// NeuroPLC — Auto-generated IEC 61131-3 SCL
// Graph: kan | Target: S71200Backend
// Work memory: 75KB | LUT points: 15
// Nodes: 11 | Ops: {'matmul': 3, 'standard_act': 2, 'bspline_lut': 2, 'add': 2, 'softmax': 1, 'argmax': 1}


DATA_BLOCK "NeuroPLC_Weights"
{ S7_Optimized_Access := 'FALSE' }
VERSION : 0.1
NON_RETAIN
   STRUCT

   // BsplineLUT 'l0_bspline': grid(15 pts) + table(16×28×15)
   w0 : ARRAY[0..14] OF REAL :=
[-3.0000000, -2.5714286, -2.1428571, -1.7142857, -1.2857143, -0.8571429, -0.4285714, 0.0
    0.4285714, 0.8571429, 1.2857143, 1.7142857, 2.1428571, 2.5714286, 3.0000000];
   w1 : ARRAY[0..6719] OF REAL :=
[-0.1678985, -0.1780923, -0.1814521, -0.1775268, -0.1656160, -0.1449310, -0.1146830, -0.0740834
    -0.0224071, 0.0378880, 0.0997435, 0.1557420, 0.1984661, 0.2204984, 0.2159406, -0.0068030
    -0.0092832, -0.0059920, 0.0046129, 0.0216460, 0.0433637, 0.0680215, 0.0938751, 0.1191888
    0.1426669, 0.1636497, 0.1815270, 0.1956886, 0.2055246, 0.2105588, -0.1221549, -0.1171233
    -0.0966766, -0.0587330, -0.0074782, 0.0506872, 0.1093601, 0.1621373, 0.2026832, 0.2280267
    0.2400602, 0.2410554, 0.2332843, 0.2190189, 0.2004736, -0.1071566, -0.1184995, -0.1260945
    -0.1291901, -0.1269063, -0.1183174, -0.1024977, -0.0785217, -0.0455032, -0.0045367, 0.0404215
    0.0851916, 0.1255936, 0.1574478, 0.1771163, -0.2579331, -0.2737922, -0.2772716, -0.2656087
    -0.2406511, -0.2058749, -0.1647583, -0.1207793, -0.0773919, -0.0368323, 0.0004230, 0.0340346
    0.0636633, 0.0889699, 0.1095319, -0.0785050, -0.0811057, -0.0777832, -0.0686172, -0.0542267
    -0.0354211, -0.0130104, 0.0121958, 0.0393740, 0.0670212, 0.0926518, 0.1137036, 0.1276142
    0.1318216, 0.1243265, 0.1783668, 0.2024992, 0.2205571, 0.2295309, 0.2281837, 0.2159047
    0.1920838, 0.1561110, 0.1074165, 0.0474421, -0.0194626, -0.0887214, -0.1557577, -0.2159953
    -0.2651629, -0.0098763, -0.0567750, -0.0900950, -0.1037325, -0.0997373, -0.0830403, -0.0585757
    -0.0312776, -0.0060409, 0.0142129, 0.0294136, 0.0397139, 0.0452663, 0.0462234, 0.0427955
    -0.1445924, -0.1514427, -0.1456748, -0.1261707, -0.0959553, -0.0595173, -0.0213470, 0.0140651
    0.0422729, 0.0610472, 0.0713624, 0.0744433, 0.0715144, 0.0638003, 0.0524706, 0.0649802
    0.0350223, 0.0192966, 0.0229814, 0.0440583, 0.0779662, 0.1201407, 0.1660179, 0.2110452
    0.2512608, 0.2835559, 0.3048884, 0.3122162, 0.3024972, 0.2736655, 0.2887279, 0.2531290
    0.2083726, 0.1575631, 0.1047861, 0.0544741, 0.0110598, -0.0210238, -0.0374280, -0.0380050
    -0.0286788, -0.0158475, -0.0059090, -0.0052614, -0.0190888, 0.0978082, 0.0375382, -0.0283595
    -0.0966197, -0.1622492, -0.2196440, -0.2631995, -0.2873112, -0.2864807, -0.2605327, -0.2169844
    -0.1639538, -0.1095588, -0.0619172, -0.0280842, 0.3787996, 0.3042307, 0.2275823, 0.1533788
    0.0834056, 0.0184802, -0.0405809, -0.0929614, -0.1378582, -0.1751406, -0.2056495, -0.2303015
    -0.2500134, -0.2657017, -0.2780562, 0.1412515, 0.1458592, 0.1559898, 0.1722250, 0.1933805
    0.2176485, 0.2432202, 0.2682872, 0.2910532, 0.3103575, 0.3259565, 0.3376784, 0.3453514
    0.3488037, 0.3478512, 0.0779829, 0.0010007, -0.0646528, -0.1104959, -0.1384850, -0.1542647
    -0.1634839, -0.1717914, -0.1847575, -0.2040232, -0.2255503, -0.2448578, -0.2574643, -0.2588886
    -0.2455201, -0.0444734, -0.0539526, -0.0628650, -0.0722421, -0.0807835, -0.0863650, -0.0868614
    -0.0801473, -0.0641548, -0.0396736, -0.0116243, 0.0147505, 0.0342076, 0.0415045, 0.0324876
    -0.0761592, -0.0368462, 0.0081775, 0.0553801, 0.1025478, 0.1479322, 0.1897853, 0.2263595
    0.2559171, 0.2772311, 0.2898127, 0.2932306, 0.2870536, 0.2708503, 0.2446318, 0.0232008
    0.0053789, -0.0155840, -0.0376546, -0.0582679, -0.0746713, -0.0841116, -0.0838361, -0.0711388
    -0.0456730, -0.0105014, 0.0310470, 0.0756434, 0.1199589, 0.1607804, 0.3611427, 0.2999726
    0.2319509, 0.1606371, 0.0886557, 0.0183016, -0.0481310, -0.1083478, -0.1600664, -0.2015907
    -0.2320727, -0.2507303, -0.2567816, -0.2494446, -0.2283804, 0.2381873, 0.2065935, 0.1685599
    0.1238492, 0.0745029, 0.0233678, -0.0267086, -0.0728783, -0.1123279, -0.1439519, -0.1691131
    -0.1893671, -0.2062695, -0.2213760, -0.2358772, -0.2661355, -0.2041683, -0.1454980, -0.0950915
    -0.0516159, -0.0115122, 0.0287810, 0.0728252, 0.1241262, 0.1833983, 0.2473215, 0.3122611
    0.3745819, 0.4306494, 0.4769619, -0.0463834, -0.0837121, -0.1064505, -0.1077356, -0.0899888
    -0.0589119, -0.0202105, 0.0204099, 0.0572939, 0.0873028, 0.1109346, 0.1289717, 0.1421960
    0.1513896, 0.1572272, -0.0369839, 0.0175120, 0.0567876, 0.0736601, 0.0717070, 0.0583079
    0.0408467, 0.0267074, 0.0231900, 0.0333957, 0.0543573, 0.0826338, 0.1147841, 0.1473674
    0.1771034, 0.0579601, 0.0613396, 0.0567427, 0.0438791, 0.0253106, 0.0046067, -0.0146619
    -0.0289245, -0.0346569, -0.0306635, -0.0191136, -0.0024393, 0.0169272, 0.0365540, 0.0541844
    0.2344523, 0.1852709, 0.1321315, 0.0796445, 0.0306498, -0.0126383, -0.0480064, -0.0732409
    -0.0861622, -0.0862884, -0.0755912, -0.0562338, -0.0303795, -0.0001915, 0.0321418, -0.3219349
    -0.2878197, -0.2440139, -0.1914641, -0.1323293, -0.0691967, -0.0046544, 0.0587098, 0.1183154
    0.1719484, 0.2179248, 0.2546021, 0.2803375, 0.2934885, 0.2928481, 0.1365492, 0.0991861
    0.0671679, 0.0442195, 0.0300286, 0.0228570, 0.0209643, 0.0226107, 0.0260721, 0.0304366
    0.0359652, 0.0430108, 0.0519260, 0.0630637, 0.0765354, 0.2151295, 0.2080802, 0.1835975
    0.1377589, 0.0763824, 0.0087284, -0.0559392, -0.1083561, -0.1393775, -0.1458259, -0.1331474
    -0.1074616, -0.0748881, -0.0415463, -0.0129262, -0.1535066, -0.1489179, -0.1361766, -0.1134237
    -0.0816039, -0.0426522, 0.0014951, 0.0489018, 0.0976467, 0.1465670, 0.1955956, 0.2447508
    0.2940510, 0.3435148, 0.3928187, -0.1842766, -0.1725566, -0.1530151, -0.1261257, -0.0929481
    -0.0547494, -0.0127967, 0.0316428, 0.0773057, 0.1231240, 0.1683109, 0.2121023, 0.2537336
    0.2924404, 0.3273210, -0.3537021, -0.3697125, -0.3730848, -0.3618120, -0.3364379, -0.2984076
    -0.2491672, -0.1901629, -0.1228470, -0.0489823, 0.0292201, 0.1095140, 0.1896530, 0.2673912
    0.3403057, 0.0691459, 0.0560939, 0.0299653, -0.0117787, -0.0650165, -0.1232729, -0.1800701
    -0.2289302, -0.2634472, -0.2808101, -0.2834036, -0.2740183, -0.2554445, -0.2304725, -0.2017861
    0.3468476, 0.3770096, 0.3880946, 0.3739721, 0.3370012, 0.2825406, 0.2159522, 0.1425982
    0.0678194, -0.0041134, -0.0704748, -0.1286606, -0.1760661, -0.2100872, -0.2284960, -0.0560788
    -0.0071707, 0.0405771, 0.0816977, 0.1138511, 0.1358018, 0.1463158, 0.1441588, 0.1281473
    0.0996185, 0.0635531, 0.0252163, -0.0101268, -0.0372110, -0.0516493, -0.3198017, -0.3047755
    -0.2896692, -0.2776229, -0.2658188, -0.2493332, -0.2232402, -0.1826140, -0.1226357, -0.0438484
    0.0454563, 0.1363818, 0.2200311, 0.2875079, 0.3310730, 0.2163881, 0.2115666, 0.1936969
    0.1613140, 0.1183200, 0.0705138, 0.0236961, -0.0163320, -0.0438224, -0.0556595, -0.0525330
    -0.0354296, -0.0053362, 0.0367607, 0.0893699, -0.2378380, -0.2452140, -0.2327680, -0.1957328
    -0.1394797, -0.0729626, -0.0051392, 0.0550326, 0.0987072, 0.1226663, 0.1318229, 0.1317253
    0.1279218, 0.1259604, 0.1306052, -0.2589217, -0.2554902, -0.2427067, -0.2166298, -0.1778840
    -0.1287070, -0.0713383, -0.0080176, 0.0590193, 0.1277189, 0.1962919, 0.2629692, 0.3259821
    0.3835616, 0.4338699, -0.4825098, -0.4378357, -0.3795550, -0.3085476, -0.2284881, -0.1440391
    -0.0598640, 0.0193734, 0.0890515, 0.1466455, 0.1926608, 0.2278395, 0.2529236, 0.2686552
    0.2757685, 0.0510817, 0.0267852, 0.0115559, 0.0100124, 0.0199990, 0.0369665, 0.0563629
    0.0736359, 0.0842873, 0.0865004, 0.0823345, 0.0741517, 0.0643138, 0.0551828, 0.0488068
    -0.3000423, -0.2227166, -0.1399772, -0.0564061, 0.0242198, 0.0984080, 0.1626662, 0.2135022
    0.2474917, 0.2646081, 0.2697350, 0.2681393, 0.2650878, 0.2658477, 0.2746548, -0.3707289
    -0.3179955, -0.2547265, -0.1827821, -0.1066126, -0.0315833, 0.0369392, 0.0935883, 0.1330773
    0.1541022, 0.1611157, 0.1590200, 0.1527170, 0.1471089, 0.1463268, -0.0303282, -0.0316194
    -0.0313303, -0.0258615, -0.0176743, -0.0113720, -0.0115601, -0.0228442, -0.0497415, -0.0923469
    -0.1443644, -0.1989989, -0.2494552, -0.2889386, -0.3116082, 0.1333115, 0.1672112, 0.1852771
    0.1834520, 0.1631691, 0.1278019, 0.0807259, 0.0253167, -0.0350523, -0.0971276, -0.1578280
    -0.2140861, -0.2628341, -0.3010046, -0.3259561, 0.3146413, 0.2845448, 0.2375658, 0.1752124
    0.1014613, 0.0211616, -0.0608367, -0.1396836, -0.2105710, -0.2707883, -0.3206561, -0.3607319
    -0.3915728, -0.4137364, -0.4276623, -0.2953075, -0.2395135, -0.1840440, -0.1340918, -0.0906518
    -0.0532361, -0.0213547, 0.0054823, 0.0277453, 0.0449382, 0.0551681, 0.0564328, 0.0467301
    0.0240579, -0.0127231, -0.3443950, -0.2914325, -0.2230571, -0.1379327, -0.0423431, 0.0547353
    0.1443230, 0.2174405, 0.2652062, 0.2836330, 0.2758078, 0.2453697, 0.1959578, 0.1312112
    0.0552579, -0.5969847, -0.5568496, -0.4988820, -0.4225912, -0.3306850, -0.2270015, -0.1153800
    0.0003402, 0.1162943, 0.2273436, 0.3265080, 0.4066636, 0.4606866, 0.4814535, 0.4636622
    0.4240763, 0.3780873, 0.3254954, 0.2679662, 0.2064849, 0.1417967, 0.0746462, 0.0057781
    -0.0640220, -0.1319213, -0.1921286, -0.2386218, -0.2653784, -0.2663764, -0.2372068, 0.3549311
    0.2616640, 0.1653353, 0.0727070, -0.0142901, -0.0954316, -0.1704954, -0.2392592, -0.3014889
    -0.3563516, -0.4021494, -0.4371169, -0.4594885, -0.4674988, -0.4598311, 0.2618391, 0.2260382
    0.1761623, 0.1113720, 0.0344484, -0.0505477, -0.1395543, -0.2285095, -0.3133526, -0.3901000
    -0.4548796, -0.5038275, -0.5330802, -0.5387741, -0.5180939, 0.1146218, 0.0686993, 0.0261798
    -0.0089268, -0.0355121, -0.0534927, -0.0627863, -0.0633110, -0.0549970, -0.0383974, -0.0149654
    0.0137755, 0.0463018, 0.0810901, 0.1164729, 0.0417326, 0.0411822, 0.0355795, 0.0236865
    0.0051303, -0.0201561, -0.0522397, -0.0911871, -0.1370274, -0.1879016, -0.2392222, -0.2861886
    -0.3240004, -0.3478571, -0.3537749, 0.3919963, 0.3451138, 0.2737949, 0.1739022, 0.0532871
    -0.0759618, -0.2017516, -0.3119893, -0.3947308, -0.4454888, -0.4705520, -0.4770510, -0.4721161
    -0.4628775, -0.4554293, -0.0126168, -0.0509731, -0.0831967, -0.1066613, -0.1219576, -0.1308127
    -0.1349550, -0.1361129, -0.1360037, -0.1357924, -0.1358456, -0.1364676, -0.1379626, -0.1406350
    -0.1446051, 0.2584295, 0.1992141, 0.1407706, 0.0851690, 0.0331316, -0.0150953, -0.0592658
    -0.0991342, -0.1344641, -0.1654932, -0.1931442, -0.2183931, -0.2422161, -0.2655895, -0.2890680
    0.1814504, 0.1560406, 0.1238631, 0.0846020, 0.0413235, -0.0017105, -0.0402371, -0.0699933
    -0.0867895, -0.0901119, -0.0847588, -0.0759432, -0.0688782, -0.0687767, -0.0798079, 0.2167516
    0.2200129, 0.2198452, 0.2137589, 0.2003766, 0.1787147, 0.1477895, 0.1066176, 0.0542793
    -0.0069583, -0.0702222, -0.1282799, -0.1738986, -0.1998461, -0.2001815, 0.3418077, 0.3005003
    0.2533219, 0.2024476, 0.1507898, 0.1015218, 0.0578167, 0.0228482, -0.0002539, -0.0105333
    -0.0101751, -0.0016098, 0.0127324, 0.0304209, 0.0491649, 0.0084501, 0.0182875, 0.0334012
    0.0528385, 0.0750525, 0.0982866, 0.1207838, 0.1407871, 0.1565614, 0.1674692, 0.1744586
    0.1786018, 0.1809709, 0.1826379, 0.1844059, 0.1765064, 0.2196629, 0.2448905, 0.2446444
    0.2216758, 0.1823734, 0.1331302, 0.0803391, 0.0303612, -0.0120419, -0.0444194, -0.0645012
    -0.0700173, -0.0586974, -0.0290885, 0.0325744, -0.0001235, -0.0308025, -0.0574152, -0.0786708
    -0.0935458, -0.1010169, -0.1000610, -0.0896901, -0.0706827, -0.0463699, -0.0202822, 0.0040500
    0.0230964, 0.0337703, -0.0545263, -0.0683008, -0.0850943, -0.1062798, -0.1300055, -0.1532799
    -0.1731101, -0.1865034, -0.1905247, -0.1851252, -0.1744277, -0.1628807, -0.1549326, -0.1550320
    -0.1666709, 0.1232095, 0.0887160, 0.0601212, 0.0408368, 0.0302367, 0.0262682, 0.0268770
    0.0300090, 0.0336161, 0.0359655, 0.0357802, 0.0318186, 0.0228393, 0.0076005, -0.0147278
    0.2201795, 0.2253740, 0.2172903, 0.1919017, 0.1522543, 0.1038936, 0.0523679, 0.0032255
    -0.0380339, -0.0683450, -0.0881606, -0.0982082, -0.0992153, -0.0919093, -0.0771561, -0.0447728
    -0.0640291, -0.0828933, -0.1010502, -0.1166342, -0.1272313, -0.1304274, -0.1238081, -0.1050070
    -0.0740562, -0.0344543, 0.0100294, 0.0556256, 0.0985653, 0.1354940, -0.1179619, -0.0810167
    -0.0497815, -0.0275970, -0.0124455, -0.0004163, 0.0124039, 0.0299280, 0.0560133, 0.0917222
    0.1340779, 0.1797886, 0.2255621, 0.2681066, 0.3042721, -0.1272539, -0.1083060, -0.0797053
    -0.0391874, 0.0101826, 0.0634562, 0.1156826, 0.1619112, 0.1972416, 0.2192794, 0.2292528
    0.2286728, 0.2190502, 0.2018959, 0.1787229, 0.1126120, 0.1354389, 0.1525481, 0.1626929
    0.1662377, 0.1641164, 0.1572638, 0.1466143, 0.1330899, 0.1169858, 0.0976906, 0.0745224
    0.0467991, 0.0138388, -0.0245556, -0.2130979, -0.2165407, -0.2060983, -0.1792987, -0.1401104
    -0.0947774, -0.0495465, -0.0106644, 0.0157041, 0.0274952, 0.0285724, 0.0232618, 0.0158893
    0.0107810, 0.0115579, 0.0891590, 0.1140725, 0.1352188, 0.1521983, 0.1640686, 0.1696956
    0.1679449, 0.1576822, 0.1378004, 0.1085657, 0.0722279, 0.0311922, -0.0121365, -0.0553532
    -0.0961057, 0.1578736, 0.1729503, 0.1827859, 0.1860957, 0.1827528, 0.1730394, 0.1572379
    0.1356310, 0.1085122, 0.0767250, 0.0419077, 0.0057608, -0.0300154, -0.0637205, -0.0937200
    0.1219553, 0.1204909, 0.1111442, 0.0926814, 0.0665890, 0.0353152, 0.0013086, -0.0329816
    -0.0651094, -0.0927796, -0.1139141, -0.1264520, -0.1283324, -0.1174944, -0.0926047, -0.3210574
    -0.2989046, -0.2712918, -0.2394569, -0.2041107, -0.1657779, -0.1249830, -0.0822503, -0.0381294
    0.0055785, 0.0452625, 0.0771708, 0.0975514, 0.1026523, 0.0896807, 0.3200986, 0.2807284
    0.2284062, 0.1641834, 0.0906839, 0.0110872, -0.0714266, -0.1536772, -0.2324955, -0.3052692
    -0.3701901, -0.4255132, -0.4694930, -0.5003846, -0.5167131, -0.1748312, -0.1799129, -0.1605858
    -0.1114278, -0.0414540, 0.0352193, 0.1044700, 0.1521760, 0.1644143, 0.1372339, 0.0810951
    0.0075831, -0.0717166, -0.1452187, -0.2027312, -0.3041509, -0.2639937, -0.2150850, -0.1581814
    -0.0940170, -0.0233181, 0.0531893, 0.1347787, 0.2206823, 0.3080428, 0.3909831, 0.4633908
    0.5191528, 0.5521570, 0.5574339, 0.0965330, 0.0451092, 0.0023842, -0.0276105, -0.0455321
    -0.0536940, -0.0544114, -0.0499998, -0.0427504, -0.0337479, -0.0223328, -0.0077097, 0.0109168
    0.0343421, 0.0629047, -0.0030185, -0.0198640, -0.0314239, -0.0331272, -0.0253625, -0.0102703
    0.0100064, 0.0333250, 0.0575613, 0.0815243, 0.1053716, 0.1293659, 0.1537700, 0.1788468
    0.2045315, -0.3042292, -0.2481812, -0.1946689, -0.1476865, -0.1072513, -0.0719759, -0.0404710
    -0.0113473, 0.0167654, 0.0442961, 0.0703129, 0.0937775, 0.1136519, 0.1288979, 0.1386143
    -0.1048548, -0.1008864, -0.0997962, -0.1004730, -0.1017998, -0.1026578, -0.1019281, -0.0984919
    -0.0912440, -0.0797672, -0.0646386, -0.0465128, -0.0260444, -0.0038881, 0.0191783, -0.0939790
    -0.0398485, 0.0127617, 0.0593301, 0.0980469, 0.1280599, 0.1485184, 0.1585714, 0.1574058
    0.1460905, 0.1284148, 0.1083804, 0.0899891, 0.0772424, 0.0734226, 0.0639287, 0.0862761
    0.0959409, 0.0932695, 0.0824167, 0.0688831, 0.0581708, 0.0557819, 0.0671351, 0.0934834
    0.1300586, 0.1716228, 0.2129377, 0.2487656, 0.2744141, 0.2868718, 0.2211201, 0.1533946
    0.0863596, 0.0213453, -0.0407895, -0.0991865, -0.1529877, -0.2013294, -0.2430814, -0.2767285
    -0.3007249, -0.3135253, -0.3135841, -0.2998512, 0.3022131, 0.2637090, 0.2171172, 0.1644126
    0.1073856, 0.0477614, -0.0127350, -0.0723783, -0.1294486, -0.1824798, -0.2303725, -0.2720563
    -0.3064606, -0.3325149, -0.3492050, 0.3392466, 0.3126993, 0.2714594, 0.2146510, 0.1455293
    0.0688093, -0.0107926, -0.0885596, -0.1597984, -0.2209733, -0.2702214, -0.3058107, -0.3260089
    -0.3290841, -0.3139513, 0.3067191, 0.2591372, 0.2119206, 0.1692937, 0.1304451, 0.0927841
    0.0537179, 0.0106537, -0.0389403, -0.0945411, -0.1512107, -0.2036668, -0.2466268, -0.2748083
    -0.2838474, 0.1625653, 0.1415380, 0.1123944, 0.0749316, 0.0320777, -0.0121329, -0.0536643
    -0.0884808, -0.1126109, -0.1252995, -0.1304398, -0.1322882, -0.1351006, -0.1431335, -0.1597394
    0.5166554, 0.5215591, 0.4949956, 0.4327331, 0.3412310, 0.2307273, 0.1114637, -0.0063177
    -0.1124656, -0.2013636, -0.2739490, -0.3316710, -0.3759787, -0.4083213, -0.4298892, 0.1351729
    0.1269306, 0.1250641, 0.1320221, 0.1440110, 0.1550311, 0.1590802, 0.1501562, 0.1223698
    0.0754777, 0.0173960, -0.0433222, -0.0981235, -0.1384550, -0.1571404, 0.3327708, 0.3185382
    0.3052332, 0.2953537, 0.2875125, 0.2789499, 0.2669047, 0.2486153, 0.2213666, 0.1847521
    0.1417018, 0.0954064, 0.0490564, 0.0058424, -0.0312945, 0.1765392, 0.1838493, 0.1913348
    0.1987953, 0.2042284, 0.2049950, 0.1984554, 0.1819698, 0.1529608, 0.1119811, 0.0641066
    0.0147661, -0.0306112, -0.0665965, -0.0886083, 0.3272812, 0.3066857, 0.2636611, 0.1950108
    0.1051633, 0.0012415, -0.1096290, -0.2203221, -0.3237405, -0.4142143, -0.4881364, -0.5420610
    -0.5725418, -0.5761332, -0.5504896, 0.2278051, 0.2094044, 0.1705757, 0.1099797, 0.0357921
    -0.0404488, -0.1072012, -0.1529231, -0.1662461, -0.1444863, -0.0975110, -0.0361671, 0.0286983
    0.0862383, 0.1270917, -0.1655097, -0.1719809, -0.1668263, -0.1452783, -0.1086140, -0.0602463
    -0.0035905, 0.0579380, 0.1209348, 0.1825338, 0.2406473, 0.2932485, 0.3383102, 0.3738059
    0.3978944, -0.2981057, -0.2943176, -0.2839422, -0.2664428, -0.2405757, -0.2048473, -0.1577640
    -0.0978318, -0.0236287, 0.0626850, 0.1537709, 0.2418867, 0.3192897, 0.3782378, 0.4121280
    -0.1586868, -0.1489341, -0.1283361, -0.0939585, -0.0484726, 0.0034693, 0.0572128, 0.1081034
    0.1515276, 0.1849213, 0.2086818, 0.2234378, 0.2298178, 0.2284506, 0.2200290, -0.1252231
    -0.0967453, -0.0594933, -0.0122600, 0.0401879, 0.0909722, 0.1332126, 0.1600285, 0.1646609
    0.1464161, 0.1133667, 0.0742698, 0.0378823, 0.0129611, 0.0068023, 0.0834799, 0.1379879
    0.1843656, 0.2200514, 0.2444678, 0.2577389, 0.2599891, 0.2513433, 0.2319673, 0.2040831
    0.1728844, 0.1437972, 0.1222471, 0.1136601, 0.1222135, -0.0542189, -0.0593817, -0.0501164
    -0.0211112, 0.0238372, 0.0777129, 0.1334966, 0.1841690, 0.2227778, 0.2457306, 0.2542909
    0.2501011, 0.2348035, 0.2100408, 0.1775758, 0.3034255, 0.2780464, 0.2463558, 0.2100950
    0.1711902, 0.1316324, 0.0934130, 0.0585232, 0.0289297, 0.0053711, -0.0131885, -0.0279235
    -0.0400085, -0.0506181, -0.0606517, -0.3965884, -0.3682756, -0.3285228, -0.2775177, -0.2172121
    -0.1501812, -0.0790007, -0.0062465, 0.0655068, 0.1337557, 0.1960984, 0.2501415, 0.2934912
    0.3237541, 0.3389650, 0.1608326, 0.1162827, 0.0624275, 0.0022430, -0.0599907, -0.1195326
    -0.1716412, -0.2115750, -0.2346503, -0.2390736, -0.2272283, -0.2018240, -0.1655702, -0.1211765
    -0.0713665, -0.3572540, -0.3305627, -0.2893769, -0.2325372, -0.1630612, -0.0854424, -0.0041762
    0.0762423, 0.1513355, 0.2175222, 0.2725155, 0.3141297, 0.3401794, 0.3484788, 0.3373067
    -0.0932589, -0.0570386, -0.0183244, 0.0228229, 0.0646355, 0.1047426, 0.1407726, 0.1703541
    0.1911504, 0.2025709, 0.2065481, 0.2052115, 0.2006907, 0.1951153, 0.1902788, 0.2385926
    0.2339801, 0.2315844, 0.2325340, 0.2356329, 0.2388632, 0.2402064, 0.2376440, 0.2291967
    0.2148689, 0.1975305, 0.1802754, 0.1661975, 0.1583905, 0.1592519, -0.0096166, 0.0259356
    0.0501742, 0.0577008, 0.0510389, 0.0355113, 0.0164439, -0.0008374, -0.0110618, -0.0117129
    -0.0042559, 0.0095336, 0.0278798, 0.0490069, 0.0711183, -0.1487758, -0.1132716, -0.0625716
    0.0072073, 0.0902357, 0.1772524, 0.2589920, 0.3261894, 0.3697036, 0.3866156, 0.3829981
    0.3656259, 0.3412738, 0.3167166, 0.2977738, -0.3100387, -0.2733864, -0.2253677, -0.1644953
    -0.0949510, -0.0229201, 0.0454102, 0.1038525, 0.1462843, 0.1698333, 0.1763237, 0.1679466
    0.1468932, 0.1153546, 0.0757038, -0.1434238, -0.1123590, -0.0765494, -0.0356650, 0.0091617
    0.0562813, 0.1040440, 0.1507999, 0.1949039, 0.2349571, 0.2699162, 0.2987655, 0.3204895
    0.3340726, 0.3386417, -0.5487098, -0.4984198, -0.4303651, -0.3412042, -0.2356422, -0.1212278
    -0.0055129, 0.1039506, 0.1996751, 0.2773809, 0.3374251, 0.3805267, 0.4074045, 0.4187779
    0.4155242, 0.0555172, 0.0089501, -0.0343089, -0.0731426, -0.1051932, -0.1276648, -0.1377611
    -0.1326858, -0.1097181, -0.0699352, -0.0199019, 0.0333883, 0.0829421, 0.1217659, 0.1438930
    0.2507761, 0.2815168, 0.3019036, 0.3074659, 0.2988722, 0.2786065, 0.2491549, 0.2130035
    0.1726394, 0.1305899, 0.0894411, 0.0517834, 0.0202074, -0.0026965, -0.0148557, -0.0135508
    0.0039421, 0.0348047, 0.0815681, 0.1386999, 0.1978184, 0.2505388, 0.2884759, 0.3033705
    0.2932548, 0.2652527, 0.2271982, 0.1869255, 0.1522683, 0.1299458, 0.0477580, 0.0434365
    0.0405601, 0.0394647, 0.0390808, 0.0378424, 0.0341828, 0.0265353, 0.0133655, -0.0052521
    -0.0269176, -0.0490496, -0.0690665, -0.0843869, -0.0928037, -0.0152840, 0.0008645, 0.0171957
    0.0322455, 0.0460338, 0.0591047, 0.0720030, 0.0852735, 0.0994517, 0.1146016, 0.1301063
    0.1452956, 0.1594994, 0.1720476, 0.1822992, 0.0835696, 0.0671618, 0.0535326, 0.0463969
    0.0453883, 0.0486983, 0.0545166, 0.0610332, 0.0664557, 0.0698963, 0.0717732, 0.0726070
    0.0729182, 0.0732271, 0.0737634, 0.1049449, 0.1112980, 0.1163793, 0.1205961, 0.1247603
    0.1298266, 0.1367502, 0.1464860, 0.1599555, 0.1763988, 0.1926262, 0.2052584, 0.2109159
    0.2062195, 0.1885442, 0.2000310, 0.2137095, 0.2303120, 0.2509218, 0.2733334, 0.2941791
    0.3100896, 0.3176959, 0.3136782, 0.2971869, 0.2709424, 0.2379440, 0.2011906, 0.1636813
    0.1281933, 0.1573572, 0.1343969, 0.1147326, 0.1017420, 0.0937354, 0.0872329, 0.0787526
    0.0648123, 0.0420057, 0.0107119, -0.0232191, -0.0535104, -0.0738849, -0.0780657, -0.0611948
    0.3010531, 0.2891479, 0.2765397, 0.2656909, 0.2555265, 0.2437214, 0.2279492, 0.2058837
    0.1752459, 0.1361346, 0.0920856, 0.0469026, 0.0043893, -0.0316503, -0.0579024, 0.1635860
    0.1539574, 0.1472781, 0.1463320, 0.1504416, 0.1577061, 0.1662235, 0.1740918, 0.1794204
    0.1809034, 0.1780789, 0.1705511, 0.1579241, 0.1398021, 0.1161234, 0.0888673, 0.0620743
    0.0338401, 0.0057287, -0.0215293, -0.0474983, -0.0717428, -0.0938275, -0.1133227, -0.1300893
    -0.1444077, -0.1565912, -0.1669530, -0.1758066, -0.1833186, 0.0159197, 0.0066792, 0.0149232
    0.0446014, 0.0900386, 0.1421585, 0.1918811, 0.2301262, 0.2479353, 0.2424391, 0.2195677
    0.1859386, 0.1481690, 0.1128762, 0.0858354, -0.0713168, -0.0199502, 0.0298431, 0.0751292
    0.1142513, 0.1460038, 0.1691816, 0.1825797, 0.1850275, 0.1770806, 0.1617894, 0.1423990
    0.1221546, 0.1043013, 0.0916331, -0.0334748, -0.0320376, -0.0298014, -0.0261495, -0.0216799
    -0.0174198, -0.0143968, -0.0136387, -0.0161503, -0.0218034, -0.0288312, -0.0353396, -0.0394340
    -0.0392202, -0.0331915, 0.1773249, 0.1659503, 0.1539691, 0.1420005, 0.1311617, 0.1227461
    0.1180473, 0.1183589, 0.1249412, 0.1373938, 0.1529160, 0.1685197, 0.1812167, 0.1880190
    0.1864402, -0.2923942, -0.2707606, -0.2375588, -0.1917769, -0.1361762, -0.0748510, -0.0118972
    0.0485893, 0.1025440, 0.1474720, 0.1831465, 0.2095181, 0.2265374, 0.2341547, 0.2324708
    -0.0474071, 0.0251755, 0.0902499, 0.1411504, 0.1772774, 0.2001740, 0.2113859, 0.2124588
    0.2049538, 0.1912038, 0.1746566, 0.1588474, 0.1473110, 0.1435826, 0.1502753, 0.1321979
    0.1203561, 0.1131415, 0.1109601, 0.1125794, 0.1161880, 0.1199738, 0.1221245, 0.1208447
    0.1151616, 0.1052926, 0.0915474, 0.0742361, 0.0536686, 0.0303347, 0.0827111, 0.0475570
    0.0205481, 0.0064576, 0.0037487, 0.0086548, 0.0174068, 0.0262355, 0.0314206, 0.0316776
    0.0292422, 0.0266253, 0.0263375, 0.0308897, 0.0422453, 0.1559601, 0.1618557, 0.1639675
    0.1625987, 0.1582690, 0.1515748, 0.1431125, 0.1334783, 0.1232918, 0.1143282, 0.1100325
    0.1139804, 0.1297475, 0.1609094, 0.2098307, 0.1285062, 0.1413710, 0.1501217, 0.1516426
    0.1458683, 0.1338110, 0.1164840, 0.0949008, 0.0700792, 0.0432541, 0.0159743, -0.0101868
    -0.0336558, -0.0528596, -0.0664548, 0.0948606, 0.1268761, 0.1429078, 0.1405430, 0.1236279
    0.0982197, 0.0703786, 0.0461643, 0.0315498, 0.0281420, 0.0312390, 0.0356463, 0.0361692
    0.0276133, 0.0058732, 0.0552858, 0.0502080, 0.0525088, 0.0651903, 0.0857229, 0.1096220
    0.1324009, 0.1495731, 0.1567168, 0.1526599, 0.1409268, 0.1254085, 0.1099961, 0.0985806
    0.0943855, 0.0418396, 0.0817039, 0.1172940, 0.1463238, 0.1689135, 0.1860333, 0.1986548
    0.2077493, 0.2142760, 0.2185863, 0.2201529, 0.2183801, 0.2126721, 0.2024331, 0.1872655
    0.4663633, 0.4355268, 0.3870336, 0.3232322, 0.2491057, 0.1705683, 0.0935353, 0.0239218
    -0.0324135, -0.0724439, -0.0972354, -0.1081735, -0.1066439, -0.0940319, -0.0719729, 0.0738696
    0.0965428, 0.1211297, 0.1485437, 0.1765138, 0.2016438, 0.2205362, 0.2297934, 0.2260842
    0.2093901, 0.1844801, 0.1564972, 0.1305842, 0.1118842, 0.1046228, 0.1359003, 0.1015587
    0.0673522, 0.0339288, 0.0038379, -0.0196987, -0.0334586, -0.0342193, -0.0188388, 0.0118115
    0.0510589, 0.0917779, 0.1268432, 0.1491292, 0.1527306, -0.1220373, -0.0604971, -0.0028596
    0.0487916, 0.0932368, 0.1295615, 0.1568516, 0.1741927, 0.1807054, 0.1772387, 0.1671403
    0.1539529, 0.1412190, 0.1324815, 0.1306253, 0.0507799, 0.0258565, -0.0043974, -0.0401240
    -0.0786176, -0.1161662, -0.1490565, -0.1735753, -0.1860673, -0.1857758, -0.1761328, -0.1608979
    -0.1438302, -0.1286890, -0.1186756, 0.2325362, 0.2295055, 0.2162579, 0.1904587, 0.1550309
    0.1147558, 0.0744166, 0.0387964, 0.0126389, -0.0013057, -0.0031671, 0.0066999, 0.0279406
    0.0602003, 0.1026374, 0.1164177, 0.0673135, 0.0136762, -0.0426207, -0.0976070, -0.1465717
    -0.1848031, -0.2075894, -0.2102974, -0.1922244, -0.1583484, -0.1140907, -0.0648728, -0.0161160
    0.0272466, 0.1381471, 0.1253827, 0.1192710, 0.1220552, 0.1312882, 0.1428656, 0.1526812
    0.1566288, 0.1506559, 0.1334072, 0.1074253, 0.0755570, 0.0406492, 0.0055486, -0.0271285
    0.0680312, 0.0441387, 0.0219850, 0.0050373, -0.0067235, -0.0145474, -0.0196863, -0.0233920
    -0.0268993, -0.0306000, -0.0336679, -0.0351812, -0.0342186, -0.0298583, -0.0212543, 0.0143462
    0.0564369, 0.0923979, 0.1172092, 0.1314177, 0.1375374, 0.1380842, 0.1355744, 0.1324771
    0.1289144, 0.1216162, 0.1070474, 0.0816731, 0.0419583, -0.0146039, 0.0458034, 0.0375886
    0.0329915, 0.0328845, 0.0373095, 0.0460150, 0.0587492, 0.0752602, 0.0952915, 0.1183475
    0.1435870, 0.1701418, 0.1971439, 0.2237252, 0.2489738, -0.0675705, -0.0779349, -0.0892847
    -0.1018459, -0.1132911, -0.1203910, -0.1199152, -0.1086332, -0.0833887, -0.0447216, 0.0014854
    0.0489326, 0.0913204, 0.1223493, 0.1366654, 0.1363059, 0.1604894, 0.1730149, 0.1692112
    0.1498870, 0.1177873, 0.0756596, 0.0262511, -0.0276837, -0.0830434, -0.1362242, -0.1835831
    -0.2214774, -0.2462641, -0.2549900, -0.0584784, -0.0510379, -0.0453863, -0.0418930, -0.0391219
    -0.0349994, -0.0274510, -0.0144024, 0.0061898, 0.0348083, 0.0696802, 0.1088568, 0.1503891
    0.1923286, 0.2326227, -0.4725194, -0.4550803, -0.4159488, -0.3504955, -0.2650665, -0.1698862
    -0.0751833, 0.0088134, 0.0719969, 0.1103557, 0.1286876, 0.1324779, 0.1272120, 0.1183756
    0.1108190, -0.0580407, -0.0716919, -0.0771220, -0.0708079, -0.0542702, -0.0308122, -0.0037389
    0.0236447, 0.0480749, 0.0683585, 0.0862949, 0.1039172, 0.1232585, 0.1463517, 0.1745565
    -0.1139666, -0.1009195, -0.0615193, 0.0101379, 0.1046543, 0.2072248, 0.3030380, 0.3772829
    0.4153398, 0.4121848, 0.3766607, 0.3186933, 0.2482083, 0.1751314, 0.1084884, -0.3386503
    -0.2988836, -0.2520140, -0.1994287, -0.1442256, -0.0901074, -0.0407772, 0.0000617, 0.0287629
    0.0445271, 0.0506694, 0.0508261, 0.0486337, 0.0477283, 0.0511901, -0.0937131, -0.0158989
    0.0475020, 0.0900333, 0.1133672, 0.1220482, 0.1206241, 0.1136427, 0.1056101, 0.0989486
    0.0930689, 0.0871467, 0.0803574, 0.0718768, 0.0610300, 0.1474761, 0.1859243, 0.2155211
    0.2335537, 0.2385381, 0.2294242, 0.2051623, 0.1647029, 0.1070674, 0.0348320, -0.0442895
    -0.1221825, -0.1907323, -0.2418242, -0.2686586, 0.2542709, 0.2512925, 0.2350916, 0.2048720
    0.1630291, 0.1130858, 0.0585664, 0.0029951, -0.0501248, -0.0983384, -0.1407059, -0.1764061
    -0.2046175, -0.2245187, -0.2353762, -0.2790252, -0.2515094, -0.2084679, -0.1471647, -0.0717860
    0.0110360, 0.0946665, 0.1724704, 0.2378644, 0.2868490, 0.3191584, 0.3348185, 0.3338551
    0.3162940, 0.2826756, 0.2748486, 0.2728063, 0.2621618, 0.2451437, 0.2223791, 0.1939294
    0.1598549, 0.1202163, 0.0751019, 0.0259923, -0.0236204, -0.0700867, -0.1097573, -0.1389828
    -0.1546804, -0.2623799, -0.2054985, -0.1354963, -0.0521019, 0.0400954, 0.1347880, 0.2256666
    0.3064217, 0.3707773, 0.4141263, 0.4342729, 0.4292103, 0.3969309, 0.3354278, 0.2440885
    0.1392560, 0.1162300, 0.0964252, 0.0810994, 0.0696869, 0.0609776, 0.0537605, 0.0468247
    0.0389880, 0.0305027, 0.0236943, 0.0210503, 0.0250582, 0.0382052, 0.0621977, 0.1259315
    0.1096482, 0.0875181, 0.0581287, 0.0236383, -0.0125329, -0.0469632, -0.0762311, -0.0969535
    -0.1076879, -0.1097951, -0.1048552, -0.0944481, -0.0801536, -0.0635219, 0.2101911, 0.1560738
    0.0989987, 0.0431247, -0.0091678, -0.0561267, -0.0960009, -0.1270391, -0.1475136, -0.1568758
    -0.1562811, -0.1470178, -0.1303744, -0.1076393, -0.0802330, -0.0709978, -0.0563350, -0.0357067
    -0.0128466, 0.0108368, 0.0347564, 0.0583261, 0.0809597, 0.1020719, 0.1211274, 0.1376621
    0.1512178, 0.1613361, 0.1675588, 0.1694942, 0.1224296, 0.1043274, 0.0855731, 0.0694867
    0.0561944, 0.0446940, 0.0339819, 0.0230546, 0.0109156, -0.0030746, -0.0190398, -0.0370635
    -0.0572292, -0.0796205, -0.1040558, -0.0767903, -0.1393753, -0.1880802, -0.2176469, -0.2287871
    -0.2243221, -0.2070753, -0.1798703, -0.1455360, -0.1071745, -0.0682824, -0.0323871, -0.0030160
    0.0163035, 0.0227576, -0.0137194, 0.0050569, 0.0242377, 0.0420958, 0.0577960, 0.0708180
    0.0806417, 0.0867471, 0.0886291, 0.0865180, 0.0817078, 0.0755753, 0.0694973, 0.0648508
    0.0627691, 0.5899228, 0.5530820, 0.4900197, 0.3984393, 0.2863394, 0.1653566, 0.0471317
    -0.0566946, -0.1346190, -0.1820228, -0.2042359, -0.2073654, -0.1975180, -0.1808006, -0.1627267
    0.0027698, 0.0031818, 0.0082551, 0.0186404, 0.0351286, 0.0585600, 0.0897753, 0.1296150
    0.1788560, 0.2350957, 0.2913363, 0.3402212, 0.3743939, 0.3864978, 0.3706397, -0.0025321
    0.0205917, 0.0429694, 0.0624773, 0.0793088, 0.0944761, 0.1089923, 0.1238704, 0.1400876
    0.1568265, 0.1706758, 0.1780221, 0.1752515, 0.1587505, 0.1258989, 0.0653871, 0.1041137
    0.1299338, 0.1369698, 0.1280959, 0.1092785, 0.0864875, 0.0656929, 0.0527867, 0.0497712
    0.0530262, 0.0584930, 0.0621127, 0.0598263, 0.0482771, 0.2008938, 0.2139753, 0.2194843
    0.2154537, 0.2038885, 0.1881971, 0.1717893, 0.1580751, 0.1504253, 0.1502483, 0.1561170
    0.1663828, 0.1793971, 0.1935114, 0.2071681, 0.1853853, 0.2319104, 0.2758777, 0.3132807
    0.3417447, 0.3594712, 0.3646623, 0.3555205, 0.3302888, 0.2892609, 0.2356933, 0.1730742
    0.1048913, 0.0346328, -0.0345319, 0.2946110, 0.2887431, 0.2792968, 0.2666786, 0.2517614
    0.2355833, 0.2191820, 0.2035956, 0.1898666, 0.1792673, 0.1734019, 0.1739004, 0.1823929
    0.2005095, 0.2291908, 0.1584648, 0.1666528, 0.1783353, 0.1939631, 0.2109868, 0.2257967
    0.2347820, 0.2343319, 0.2208878, 0.1935178, 0.1550855, 0.1087505, 0.0576728, 0.0050121
    -0.0461847, 0.1433635, 0.1457650, 0.1450598, 0.1404541, 0.1326062, 0.1226875, 0.1118699
    0.1013256, 0.0922152, 0.0851375, 0.0798789, 0.0761625, 0.0737114, 0.0722486, 0.0715160
    0.0642120, 0.0710823, 0.0799319, 0.0885070, 0.0971988, 0.1073328, 0.1202358, 0.1372344
    0.1596237, 0.1871156, 0.2171343, 0.2469256, 0.2737350, 0.2948082, 0.3077406, 0.0792082
    0.0430626, 0.0187277, 0.0104475, 0.0159365, 0.0306019, 0.0498483, 0.0690801, 0.0837509
    0.0917590, 0.0945363, 0.0937904, 0.0912291, 0.0885601, 0.0872292, -0.0366219, -0.0059975
    0.0211352, 0.0437861, 0.0615249, 0.0741193, 0.0813369, 0.0829455, 0.0787241, 0.0690206
    0.0550045, 0.0379096, 0.0189697, -0.0005816, -0.0195318, 0.1408100, 0.1453754, 0.1567995
    0.1752028, 0.1973212, 0.2186946, 0.2348618, 0.2413613, 0.2338025, 0.2113334, 0.1782158
    0.1391110, 0.0986801, 0.0615845, 0.0318855, 0.3728876, 0.3636605, 0.3531002, 0.3411653
    0.3270430, 0.3096478, 0.2878939, 0.2606955, 0.2269944, 0.1871089, 0.1433476, 0.0981741
    0.0540520, 0.0134451, -0.0214319, 0.2175054, 0.2198412, 0.2244289, 0.2304279, 0.2359889
    0.2389059, 0.2369727, 0.2279830, 0.2097863, 0.1830311, 0.1524101, 0.1229322, 0.0996059
    0.0874400, 0.0903775, 0.2911958, 0.2672293, 0.2417178, 0.2170962, 0.1953312, 0.1782237
    0.1675746, 0.1651847, 0.1727999, 0.1894183, 0.2100667, 0.2294619, 0.2423206, 0.2433596
    0.2283258, 0.3827878, 0.3411886, 0.2981977, 0.2569056, 0.2171632, 0.1776772, 0.1371527
    0.0942950, 0.0478225, -0.0028898, -0.0575175, -0.1156620, -0.1769250, -0.2409081, -0.3066716
    0.2251391, 0.2507458, 0.2758858, 0.2986796, 0.3178295, 0.3322430, 0.3408278, 0.3424918
    0.3361631, 0.3217956, 0.3008249, 0.2748025, 0.2452798, 0.2138081, 0.1819130, 0.1689708
    0.1711256, 0.1707270, 0.1694824, 0.1680544, 0.1667367, 0.1658224, 0.1656048, 0.1663845
    0.1688381, 0.1741858, 0.1836898, 0.1986126, 0.2202167, 0.2490858, 0.1198459, 0.1158715
    0.1187188, 0.1281465, 0.1421744, 0.1582081, 0.1736523, 0.1859118, 0.1924255, 0.1923409
    0.1872750, 0.1790374, 0.1694379, 0.1602861, 0.1530649, 0.2813690, 0.2857699, 0.2775994
    0.2518772, 0.2097207, 0.1544021, 0.0891956, 0.0173756, -0.0577623, -0.1318692, -0.1990736
    -0.2533852, -0.2888138, -0.2993691, -0.2805221, -0.0945949, -0.0859146, -0.0666549, -0.0339619
    0.0098287, 0.0605471, 0.1140217, 0.1660807, 0.2125873, 0.2511515, 0.2819078, 0.3051879
    0.3213233, 0.3306457, 0.3334457, 0.1866198, 0.1884683, 0.1787530, 0.1577976, 0.1277766
    0.0915189, 0.0518542, 0.0116119, -0.0263894, -0.0598831, -0.0874005, -0.1075351, -0.1188804
    -0.1200301, -0.1100685, -0.0816909, -0.0186953, 0.0434542, 0.1009326, 0.1520018, 0.1956610
    0.2309103, 0.2567496, 0.2721971, 0.2771671, 0.2728699, 0.2606167, 0.2417188, 0.2174875
    0.1892796, 0.1155247, 0.1110856, 0.1127015, 0.1249412, 0.1436904, 0.1617671, 0.1719855
    0.1671601, 0.1402411, 0.0909893, 0.0290077, -0.0353323, -0.0916595, -0.1296024, -0.1405761
    0.0366876, 0.0358489, 0.0423771, 0.0582548, 0.0821032, 0.1113558, 0.1434446, 0.1758020
    0.2058747, 0.2318435, 0.2529499, 0.2685182, 0.2778728, 0.2803380, 0.2754306, 0.0936999
    0.0709418, 0.0538988, 0.0490415, 0.0548760, 0.0670938, 0.0813836, 0.0934337, 0.0989831
    0.0962942, 0.0872764, 0.0741241, 0.0590313, 0.0441924, 0.0315632, 0.0454234, 0.0491984
    0.0596057, 0.0783299, 0.1034458, 0.1317532, 0.1600503, 0.1851351, 0.2038397, 0.2146847
    0.2186308, 0.2168294, 0.2104321, 0.2005902, 0.1883695, -0.0667184, -0.0664766, -0.0577000
    -0.0366789, -0.0050464, 0.0336767, 0.0759675, 0.1183029, 0.1571787, 0.1900285, 0.2156412
    0.2329118, 0.2407350, 0.2380057, 0.2240467, -0.2274597, -0.1690933, -0.1114029, -0.0583104
    -0.0110341, 0.0301627, 0.0650176, 0.0932684, 0.1146536, 0.1289366, 0.1359178, 0.1354002
    0.1271870, 0.1110814, 0.0872085, -0.1521940, -0.1380929, -0.1188272, -0.0936891, -0.0636631
    -0.0303315, 0.0047229, 0.0399170, 0.0736799, 0.1050380, 0.1338809, 0.1601658, 0.1838497
    0.2048900, 0.2230166, -0.1046155, -0.0858807, -0.0573247, -0.0168516, 0.0333484, 0.0895709
    0.1481097, 0.2052584, 0.2573313, 0.3016632, 0.3370647, 0.3624612, 0.3767782, 0.3789415
    0.3681934, 0.2072487, 0.1864112, 0.1563267, 0.1171031, 0.0715261, 0.0233276, -0.0237592
    -0.0660013, -0.0997112, -0.1234848, -0.1392170, -0.1490607, -0.1551685, -0.1596933, -0.1644943
    -0.1517255, -0.1193664, -0.0782033, -0.0303212, 0.0200548, 0.0679433, 0.1083623, 0.1363294
    0.1469480, 0.1396034, 0.1198693, 0.0938024, 0.0674594, 0.0468970, 0.0370763, 0.3110608
    0.2861295, 0.2560543, 0.2233990, 0.1888246, 0.1523195, 0.1138714, 0.0734681, 0.0311259
    -0.0117016, -0.0514840, -0.0845288, -0.1071434, -0.1156352, -0.1071404, -0.0434422, -0.0256309
    -0.0061618, 0.0137750, 0.0348048, 0.0581937, 0.0852092, 0.1171182, 0.1551570, 0.1990083
    0.2461095, 0.2937233, 0.3391118, 0.3795376, 0.4124577, 0.3129768, 0.3337277, 0.3466819
    0.3502223, 0.3445130, 0.3303478, 0.3085208, 0.2798265, 0.2450805, 0.2061687, 0.1665232
    0.1296974, 0.0992442, 0.0787167, 0.0710807, -0.1485267, -0.1266887, -0.1059538, -0.0874314
    -0.0694476, -0.0493445, -0.0244634, 0.0078547, 0.0501971, 0.1015688, 0.1557980, 0.2063088
    0.2465250, 0.2698708, 0.2709672, 0.0836342, 0.1186020, 0.1419933, 0.1506651, 0.1472868
    0.1365815, 0.1232745, 0.1120911, 0.1076754, 0.1105969, 0.1155374, 0.1167185, 0.1083621
    0.0846902, 0.0412880, 0.3746155, 0.3008116, 0.2295846, 0.1697616, 0.1228553, 0.0877933
    0.0635006, 0.0489020, 0.0429200, 0.0443591, 0.0518531, 0.0640224, 0.0794876, 0.0968693
    0.1147441, 0.2624251, 0.2889178, 0.2926807, 0.2688918, 0.2221700, 0.1604698, 0.0917496
    0.0239679, -0.0349867, -0.0807150, -0.1138608, -0.1354617, -0.1465550, -0.1481785, -0.1414872
    -0.2038390, -0.1836262, -0.1623666, -0.1409924, -0.1188838, -0.0948732, -0.0677921, -0.0364720
    0.0002305, 0.0422140, 0.0875773, 0.1342791, 0.1802779, 0.2235323, 0.2620180, 0.2164622
    0.2150818, 0.2096564, 0.2016837, 0.1911032, 0.1773035, 0.1596727, 0.1375989, 0.1105010
    0.0793446, 0.0473304, 0.0178336, -0.0057705, -0.0201069, -0.0225886, 0.1444894, 0.1318568
    0.1201072, 0.1098967, 0.1011122, 0.0933685, 0.0862802, 0.0794619, 0.0725155, 0.0644148
    0.0532257, 0.0369429, 0.0135614, -0.0189239, -0.0617012, -0.3946738, -0.3444622, -0.2891815
    -0.2324311, -0.1744639, -0.1143506, -0.0511602, 0.0160378, 0.0881280, 0.1636738, 0.2378847
    0.3057082, 0.3620918, 0.4019832, 0.4212244, -0.3757093, -0.3162996, -0.2499295, -0.1809414
    -0.1102374, -0.0375038, 0.0375741, 0.1153111, 0.1959576, 0.2765333, 0.3493883, 0.4065088
    0.4398806, 0.4414897, 0.4052696, 0.3683745, 0.3139668, 0.2502587, 0.1805291, 0.1085247
    0.0381577, -0.0266595, -0.0820146, -0.1240428, -0.1512654, -0.1656516, -0.1694398, -0.1648687
    -0.1541766, -0.1394859, -0.1072037, -0.0830137, -0.0531947, -0.0165176, 0.0251676, 0.0689225
    0.1118077, 0.1508839, 0.1832300, 0.2068588, 0.2211318, 0.2255158, 0.2194776, 0.2024842
    0.1744064, -0.3319098, -0.3459042, -0.3396719, -0.3077802, -0.2539578, -0.1851701, -0.1083861
    -0.0305750, 0.0413362, 0.1025240, 0.1512056, 0.1858353, 0.2048676, 0.2067567, 0.1907547
    0.4012429, 0.3313338, 0.2576209, 0.1851532, 0.1146888, 0.0454699, -0.0232633, -0.0922704
    -0.1622683, -0.2318351, -0.2964571, -0.3513798, -0.3918482, -0.4131078, -0.4113880, 0.0432662
    0.0463959, 0.0470551, 0.0450016, 0.0397214, 0.0306044, 0.0170404, -0.0015809, -0.0258282
    -0.0542036, -0.0822218, -0.1051644, -0.1183129, -0.1169490, -0.0974791, 0.0945418, 0.0474351
    0.0144671, -0.0002516, 0.0002686, 0.0105011, 0.0249166, 0.0379856, 0.0442405, 0.0413054
    0.0312731, 0.0165850, -0.0003173, -0.0169924, -0.0312270, 0.2655172, 0.1779016, 0.0932373
    0.0169355, -0.0501629, -0.1088321, -0.1598481, -0.2039869, -0.2420160, -0.2742825, -0.3005254
    -0.3204366, -0.3337076, -0.3400303, -0.3391558, 0.2147407, 0.1649244, 0.1186844, 0.0787383
    0.0455533, 0.0188009, -0.0018479, -0.0167224, -0.0261599, -0.0309140, -0.0323391, -0.0318368
    -0.0308084, -0.0306556, -0.0325397, 0.3099983, 0.2146933, 0.1365787, 0.0858170, 0.0575848
    0.0417632, 0.0282275, 0.0068529, -0.0323252, -0.0912628, -0.1603408, -0.2290366, -0.2868275
    -0.3231913, -0.3294227, 0.2400604, 0.2115027, 0.1766969, 0.1370982, 0.0944029, 0.0503929
    0.0068497, -0.0344446, -0.0717136, -0.1034392, -0.1284772, -0.1457126, -0.1540302, -0.1523151
    -0.1398969, -0.3239543, -0.2696758, -0.2072356, -0.1376939, -0.0635290, 0.0122797, 0.0867520
    0.1569077, 0.2197818, 0.2731606, 0.3159163, 0.3470059, 0.3653866, 0.3700153, 0.3602427
    -0.1058964, -0.1240447, -0.1388698, -0.1496570, -0.1540083, -0.1489309, -0.1314311, -0.0985154
    -0.0472808, 0.0206385, 0.0970508, 0.1732528, 0.2405411, 0.2902125, 0.3149041, -0.0809075
    -0.0761908, -0.0678088, -0.0552605, -0.0376747, -0.0140495, 0.0166171, 0.0553272, 0.1030094
    0.1569253, 0.2090360, 0.2508892, 0.2740322, 0.2700127, 0.2324689, 0.0183774, 0.0161987
    0.0196904, 0.0307010, 0.0474037, 0.0666728, 0.0853814, 0.1004023, 0.1086441, 0.1087988
    0.1021359, 0.0901261, 0.0742400, 0.0559482, 0.0367036, -0.0097957, -0.0039892, 0.0028189
    0.0105871, 0.0193478, 0.0291596, 0.0400810, 0.0521704, 0.0654758, 0.0795114, 0.0930206
    0.1046862, 0.1131914, 0.1172192, 0.1157655, 0.1191704, 0.1311087, 0.1458877, 0.1635177
    0.1823133, 0.1999896, 0.2142612, 0.2228424, 0.2234735, 0.2151740, 0.1988128, 0.1754036
    0.1459593, 0.1114936, 0.0729542, 0.1572977, 0.1453381, 0.1355189, 0.1300476, 0.1291831
    0.1324956, 0.1395545, 0.1499293, 0.1631903, 0.1789441, 0.1968503, 0.2165725, 0.2377743
    0.2601195, 0.2829789, 0.0628695, 0.0769969, 0.0860344, 0.0877927, 0.0827342, 0.0722577
    0.0577633, 0.0406512, 0.0223093, 0.0035208, -0.0158050, -0.0358270, -0.0567041, -0.0785953
    -0.1016069, 0.1131401, 0.1069956, 0.0981420, 0.0867915, 0.0734585, 0.0587646, 0.0433313
    0.0277801, 0.0127375, -0.0009211, -0.0119603, -0.0191169, -0.0211274, -0.0167287, -0.0051465
    0.0572075, 0.0357429, 0.0213811, 0.0165095, 0.0211165, 0.0343429, 0.0553284, 0.0832127
    0.1171167, 0.1552116, 0.1942961, 0.2310619, 0.2622007, 0.2844040, 0.2948321, 0.1434070
    0.1549482, 0.1670772, 0.1781332, 0.1874069, 0.1945248, 0.1991140, 0.2008018, 0.1992118
    0.1938003, 0.1837813, 0.1683501, 0.1467019, 0.1180318, 0.0819414, 0.0750777, 0.0777608
    0.0672206, 0.0439258, 0.0107293, -0.0286731, -0.0705851, -0.1113101, -0.1471814, -0.1760247
    -0.1978224, -0.2127253, -0.2208840, -0.2224495, -0.2176575, 0.1612096, 0.1444548, 0.1335241
    0.1296110, 0.1294437, 0.1281723, 0.1209451, 0.1029104, 0.0692988, 0.0194586, -0.0413110
    -0.1072460, -0.1725826, -0.2315571, -0.2789746, 0.4111212, 0.3551752, 0.2895649, 0.2152339
    0.1348414, 0.0516528, -0.0310660, -0.1100489, -0.1820429, -0.2444422, -0.2955766, -0.3338489
    -0.3576620, -0.3654186, -0.3560661, 0.1391590, 0.1250600, 0.1217095, 0.1317212, 0.1507030
    0.1717879, 0.1881056, 0.1927863, 0.1790760, 0.1460479, 0.1011956, 0.0526702, 0.0086227
    -0.0227959, -0.0347899, 0.0559819, 0.0581868, 0.0646391, 0.0766424, 0.0923719, 0.1088978
    0.1232888, 0.1326139, 0.1339891, 0.1269062, 0.1142898, 0.0993324, 0.0852266, 0.0751649
    0.0718163, 0.2732919, 0.2494898, 0.2191522, 0.1815386, 0.1363864, 0.0836023, 0.0230931
    -0.0452346, -0.1214316, -0.2034314, -0.2861067, -0.3640917, -0.4320202, -0.4845264, -0.5169412
    -0.0691999, -0.1076962, -0.1233470, -0.1107835, -0.0727259, -0.0147534, 0.0575521, 0.1386083
    0.2228317, 0.3045648, 0.3780438, 0.4374964, 0.4771504, 0.4912336, 0.4753526, -0.0001498
    -0.0032703, 0.0011039, 0.0176806, 0.0448323, 0.0786930, 0.1153941, 0.1510671, 0.1818855
    0.2061389, 0.2251743, 0.2405776, 0.2539347, 0.2668312, 0.2804183, 0.2785104, 0.2438975
    0.2035888, 0.1580865, 0.1088918, 0.0578585, 0.0068411, -0.0423062, -0.0877313, -0.1277092
    -0.1606971, -0.1851669, -0.1995904, -0.2024393, -0.1926829, 0.4454534, 0.3676981, 0.2863407
    0.2065850, 0.1303759, 0.0585069, -0.0082298, -0.0690421, -0.1231326, -0.1694447, -0.2065468
    -0.2329782, -0.2472781, -0.2479858, -0.2341930, -0.2216615, -0.2067420, -0.1850035, -0.1541864
    -0.1140946, -0.0652607, -0.0082182, 0.0564991, 0.1283061, 0.2040327, 0.2767734, 0.3393309
    0.3845079, 0.4051074, 0.3954616, -0.0241830, -0.0147689, -0.0074899, -0.0015797, 0.0041061
    0.0108452, 0.0199157, 0.0325956, 0.0501315, 0.0722017, 0.0962181, 0.1194157, 0.1390292
    0.1522937, 0.1568849, -0.0959317, -0.0528233, -0.0092763, 0.0343819, 0.0779881, 0.1214369
    0.1646231, 0.2074412, 0.2497654, 0.2904309, 0.3267724, 0.3560070, 0.3753522, 0.3820254
    0.3738285, -0.0641084, -0.0609075, -0.0583547, -0.0550581, -0.0502603, -0.0434279, -0.0340281
    -0.0215279, -0.0054111, 0.0139915, 0.0351259, 0.0563423, 0.0759910, 0.0924222, 0.1041725
    -0.0341204, -0.0091993, 0.0193507, 0.0505301, 0.0828547, 0.1146690, 0.1443173, 0.1701441
    0.1905136, 0.2047915, 0.2137906, 0.2184365, 0.2196550, 0.2183718, 0.2153754, -0.0186932
    0.0193089, 0.0562244, 0.0918554, 0.1257393, 0.1573201, 0.1860417, 0.2113482, 0.2326842
    0.2495404, 0.2614738, 0.2680464, 0.2688202, 0.2633573, 0.2513908, 0.0566885, 0.1031851
    0.1373615, 0.1554016, 0.1597643, 0.1551255, 0.1461639, 0.1375579, 0.1339277, 0.1369582
    0.1440933, 0.1524456, 0.1591280, 0.1612530, 0.1563877, -0.0301588, -0.0067982, 0.0122754
    0.0251599, 0.0333866, 0.0396994, 0.0468439, 0.0575657, 0.0745624, 0.0981387, 0.1251408
    0.1521448, 0.1757269, 0.1924634, 0.1994423, 0.3237398, 0.3147339, 0.2917620, 0.2528614
    0.2016544, 0.1437367, 0.0847061, 0.0301604, -0.0143777, -0.0471586, -0.0718843, -0.0926829
    -0.1136822, -0.1390103, -0.1718136, 0.5322388, 0.4516525, 0.3699894, 0.2936842, 0.2215195
    0.1495740, 0.0739234, -0.0093567, -0.1040900, -0.2090549, -0.3157387, -0.4150598, -0.4979360
    -0.5552858, -0.5795367, 0.3348313, 0.3139692, 0.2890814, 0.2616292, 0.2314300, 0.1977201
    0.1597350, 0.1167106, 0.0679124, 0.0141103, -0.0417528, -0.0965641, -0.1472107, -0.1905800
    -0.2238805, 0.0441595, 0.0223551, 0.0117973, 0.0164633, 0.0346856, 0.0628025, 0.0971498
    0.1340633, 0.1699050, 0.2023456, 0.2309466, 0.2554175, 0.2754675, 0.2908060, 0.3011061
    0.0938526, 0.0646245, 0.0408562, 0.0255288, 0.0176385, 0.0147738, 0.0145215, 0.0144682
    0.0122432, 0.0075938, 0.0033288, 0.0024960, 0.0081430, 0.0233176, 0.0503320, -0.1736872
    -0.2018598, -0.2184409, -0.2198891, -0.2069418, -0.1818479, -0.1468583, -0.1042237, -0.0562133
    -0.0060076, 0.0418950, 0.0828932, 0.1123860, 0.1257721, 0.1194308, 0.2034807, 0.2159660
    0.2251174, 0.2297540, 0.2297332, 0.2252793, 0.2166169, 0.2039706, 0.1875626, 0.1674950
    0.1436959, 0.1160799, 0.0845618, 0.0490560, 0.0097851, 0.0084393, -0.0037575, -0.0096962
    -0.0075738, 0.0020896, 0.0179530, 0.0386746, 0.0629125, 0.0893207, 0.1163582, 0.1422011
    0.1650037, 0.1829203, 0.1941051, 0.1969572, 0.2633480, 0.2195053, 0.1743630, 0.1311768
    0.0902144, 0.0506880, 0.0118084, -0.0272136, -0.0671537, -0.1081212, -0.1492622, -0.1896475
    -0.2283478, -0.2644342, -0.2968259, -0.0753155, -0.0705651, -0.0563480, -0.0336360, -0.0058240
    0.0228373, 0.0480962, 0.0657007, 0.0714666, 0.0645810, 0.0491042, 0.0294766, 0.0101389
    -0.0044685, -0.0106460, 0.2106405, 0.1830579, 0.1505358, 0.1133623, 0.0735978, 0.0339286
    -0.0029582, -0.0343754, -0.0576678, -0.0717680, -0.0779037, -0.0774818, -0.0719092, -0.0625927
    -0.0509060, -0.3274674, -0.2629944, -0.2038490, -0.1565354, -0.1200805, -0.0908690, -0.0652826
    -0.0397029, -0.0105580, 0.0234085, 0.0601056, 0.0971813, 0.1322834, 0.1630599, 0.1873036
    -0.0690877, -0.0509122, -0.0313818, -0.0091832, 0.0158236, 0.0433644, 0.0731640, 0.1049476
    0.1384244, 0.1725134, 0.2049913, 0.2335457, 0.2558642, 0.2696344, 0.2729122, -0.0589441
    -0.0342618, -0.0055190, 0.0271774, 0.0612910, 0.0934264, 0.1201872, 0.1381771, 0.1440491
    0.1369218, 0.1194770, 0.0946747, 0.0654752, 0.0348383, 0.0055348, 0.1142520, 0.1359137
    0.1489129, 0.1481625, 0.1358423, 0.1167002, 0.0954867, 0.0769527, 0.0657870, 0.0635884
    0.0674900, 0.0742760, 0.0807309, 0.0836388, 0.0802503, -0.4963562, -0.4881529, -0.4580787
    -0.4027445, -0.3260558, -0.2344954, -0.1345493, -0.0327034, 0.0645796, 0.1520003, 0.2259398
    0.2829104, 0.3194247, 0.3319951, 0.3183341, -0.2581464, -0.2259318, -0.1867423, -0.1417929
    -0.0931570, -0.0432113, 0.0056672, 0.0511014, 0.0907371, 0.1233640, 0.1494249, 0.1694916
    0.1841360, 0.1939300, 0.1995259, 0.2516904, 0.2530169, 0.2526439, 0.2516513, 0.2490327
    0.2430442, 0.2319413, 0.2139793, 0.1874578, 0.1528830, 0.1139504, 0.0746044, 0.0387894
    0.0104499, -0.0071207, 0.2666245, 0.2363470, 0.2008183, 0.1616806, 0.1188768, 0.0717494
    0.0196403, -0.0381088, -0.1021090, -0.1706225, -0.2385168, -0.3003941, -0.3508568, -0.3845074
    -0.3969070, -0.0286634, -0.0313490, -0.0325963, -0.0315775, -0.0271991, -0.0182737, -0.0036136
    0.0179685, 0.0476130, 0.0841017, 0.1228077, 0.1588378, 0.1872988, 0.2032979, 0.2028342
    0.0822806, 0.1055830, 0.1210727, 0.1261290, 0.1226352, 0.1140661, 0.1038982, 0.0956081
    0.0926303, 0.0963046, 0.1049423, 0.1166188, 0.1294093, 0.1413890, 0.1507615, -0.2690735
    -0.1935901, -0.1172682, -0.0456560, 0.0191559, 0.0762989, 0.1249055, 0.1641084, 0.1930635
    0.2120976, 0.2232291, 0.2286085, 0.2303862, 0.2307129, 0.2313590, -0.0819909, -0.0262301
    0.0238818, 0.0636981, 0.0940510, 0.1177084, 0.1374404, 0.1560169, 0.1761686, 0.1986485
    0.2213520, 0.2419512, 0.2581182, 0.2675254, 0.2681968, -0.0461046, -0.0095733, 0.0161245
    0.0269383, 0.0255286, 0.0169270, 0.0061681, -0.0017138, -0.0017482, 0.0078269, 0.0241367
    0.0439447, 0.0640142, 0.0811086, 0.0923875, 0.1214715, 0.1246429, 0.1179697, 0.1021397
    0.0794863, 0.0529245, 0.0253697, -0.0002625, -0.0210925, -0.0360475, -0.0466648, -0.0546860
    -0.0618522, -0.0699049, -0.0802395, -0.1132871, -0.0717634, -0.0319256, 0.0041296, 0.0359250
    0.0635558, 0.0871177, 0.1067064, 0.1224124, 0.1340688, 0.1411366, 0.1430477, 0.1392339
    0.1291272, 0.1124477, 0.1065226, 0.0679530, 0.0277192, -0.0120758, -0.0494568, -0.0824937
    -0.1092565, -0.1278153, -0.1362775, -0.1346298, -0.1255739, -0.1120240, -0.0968938, -0.0830973
    -0.0731394, 0.0702876, 0.0351664, 0.0094846, -0.0018965, -0.0003208, 0.0106751, 0.0275520
    0.0467709, 0.0648162, 0.0793579, 0.0897788, 0.0955954, 0.0963241, 0.0914817, 0.0808327
    -0.1561871, -0.1465697, -0.1172424, -0.0641265, 0.0073557, 0.0884247, 0.1702974, 0.2441905
    0.3014090, 0.3376742, 0.3550895, 0.3562566, 0.3437775, 0.3202540, 0.2883357, -0.2523765
    -0.2036962, -0.1455273, -0.0788729, -0.0065118, 0.0681494, 0.1417037, 0.2107440, 0.2718817
    0.3226697, 0.3620203, 0.3889524, 0.4024845, 0.4016355, 0.3857890, -0.2730969, -0.2395672
    -0.1975484, -0.1479309, -0.0912749, -0.0280236, 0.0413795, 0.1164914, 0.1968288, 0.2799235
    0.3604371, 0.4328076, 0.4914726, 0.5308703, 0.5462435, 0.2663759, 0.2617837, 0.2487071
    0.2273422, 0.2011032, 0.1745413, 0.1522086, 0.1386574, 0.1383519, 0.1513314, 0.1712411
    0.1912272, 0.2044355, 0.2040123, 0.1844213, -0.1322568, -0.1054526, -0.0694236, -0.0246700
    0.0254581, 0.0766039, 0.1244093, 0.1645163, 0.1926105, 0.2065688, 0.2074343, 0.1964972
    0.1750481, 0.1443772, 0.1058727, 0.0963661, 0.0729697, 0.0442535, 0.0105362, -0.0263189
    -0.0639028, -0.0998057, -0.1316179, -0.1569322, -0.1734747, -0.1791631, -0.1719304, -0.1497096
    -0.1104336, -0.0529810, -0.1897976, -0.1489798, -0.1093301, -0.0766478, -0.0506775, -0.0290246
    -0.0092918, 0.0109181, 0.0339771, 0.0610016, 0.0912931, 0.1240118, 0.1583174, 0.1933700
    0.2281768, -0.0203649, -0.0136181, -0.0048761, 0.0046482, 0.0139614, 0.0221468, 0.0282883
    0.0314697, 0.0308098, 0.0271957, 0.0240692, 0.0250715, 0.0338439, 0.0540278, 0.0882226
    -0.1464982, -0.0937421, -0.0454817, -0.0063742, 0.0244465, 0.0497983, 0.0725012, 0.0953754
    0.1211933, 0.1503596, 0.1798554, 0.2063952, 0.2266930, 0.2374634, 0.2360676, 0.0611053
    0.0746875, 0.0845858, 0.0889394, 0.0865942, 0.0766460, 0.0581907, 0.0303245, -0.0078133
    -0.0549158, -0.1065438, -0.1580134, -0.2046408, -0.2417421, -0.2652695, -0.0629327, -0.0544456
    -0.0388863, -0.0146231, 0.0167074, 0.0523138, 0.0894034, 0.1251835, 0.1568739, 0.1823232
    0.2002880, 0.2095961, 0.2090753, 0.1975532, 0.1743914, 0.2462173, 0.2479595, 0.2435866
    0.2337594, 0.2202922, 0.2054069, 0.1913256, 0.1802706, 0.1744293, 0.1742365, 0.1775948
    0.1822091, 0.1857844, 0.1860255, 0.1810417, 0.1842394, 0.1759240, 0.1652069, 0.1531290
    0.1407570, 0.1291665, 0.1194330, 0.1126322, 0.1098006, 0.1100169, 0.1095305, 0.1043701
    0.0905640, 0.0641410, 0.0222768, 0.2324026, 0.2270462, 0.2092644, 0.1759481, 0.1304366
    0.0783474, 0.0253004, -0.0230842, -0.0612384, -0.0862012, -0.0987797, -0.1000750, -0.0911881
    -0.0732202, -0.0475565, -0.1538858, -0.1476419, -0.1318033, -0.1059194, -0.0719550, -0.0327286
    0.0089407, 0.0502336, 0.0883495, 0.1214252, 0.1489520, 0.1705270, 0.1857473, 0.1942100
    0.1956356, 0.1781234, 0.2150935, 0.2364076, 0.2349799, 0.2128720, 0.1753774, 0.1277933
    0.0754168, 0.0235110, -0.0243842, -0.0672181, -0.1041347, -0.1342779, -0.1567914, -0.1709817
    0.1261699, 0.1204049, 0.1132670, 0.1045704, 0.0956178, 0.0882376, 0.0842590, 0.0855112
    0.0937813, 0.1087499, 0.1270531, 0.1450896, 0.1592580, 0.1659569, 0.1621570, 0.2012317
    0.2204620, 0.2296677, 0.2267044, 0.2127215, 0.1900325, 0.1609519, 0.1277944, 0.0928715
    0.0583375, 0.0261192, -0.0018743, -0.0237338, -0.0375503, -0.0418454, -0.5280923, -0.4531125
    -0.3649584, -0.2686976, -0.1686778, -0.0689929, 0.0262637, 0.1129985, 0.1871544, 0.2464946
    0.2914124, 0.3225066, 0.3403762, 0.3456200, 0.3389946, -0.1168600, -0.0961219, -0.0717191
    -0.0456075, -0.0183319, 0.0100613, 0.0395266, 0.0700183, 0.1014772, 0.1331632, 0.1633520
    0.1902426, 0.2120339, 0.2269250, 0.2333222, 0.2793344, 0.2383755, 0.1941289, 0.1486612
    0.1042631, 0.0633041, 0.0281537, 0.0011814, -0.0153013, -0.0218949, -0.0234084, -0.0249789
    -0.0317440, -0.0488409, -0.0801608, 0.1238915, 0.0987584, 0.0669696, 0.0302128, -0.0088337
    -0.0471413, -0.0816814, -0.1094251, -0.1273871, -0.1347596, -0.1338822, -0.1273400, -0.1177180
    -0.1076013, -0.0992385, 0.3960009, 0.3587182, 0.2956125, 0.2037258, 0.0910976, -0.0303465
    -0.1486770, -0.2519639, -0.3284195, -0.3733740, -0.3924430, -0.3920458, -0.3786012, -0.3585284
    -0.3375227, 0.3986191, 0.3502203, 0.2943892, 0.2322398, 0.1662881, 0.0995453, 0.0350232
    -0.0242665, -0.0753394, -0.1165882, -0.1483954, -0.1712990, -0.1858369, -0.1925469, -0.1920198
    0.0019573, -0.0328276, -0.0593076, -0.0763549, -0.0842564, -0.0837986, -0.0757685, -0.0609534
    -0.0401386, -0.0140248, 0.0168097, 0.0517962, 0.0903661, 0.1319506, 0.1756335, 0.3860057
    0.3204645, 0.2517192, 0.1827146, 0.1138553, 0.0446483, -0.0254004, -0.0967846, -0.1699500
    -0.2429159, -0.3101957, -0.3660291, -0.4046555, -0.4203149, -0.4085274, 0.3202668, 0.2824083
    0.2450568, 0.2115314, 0.1838702, 0.1636585, 0.1524811, 0.1519227, 0.1635095, 0.1858246
    0.2131982, 0.2396286, 0.2591140, 0.2656527, 0.2543574, -0.1222956, -0.0653846, -0.0125224
    0.0309169, 0.0647700, 0.0907150, 0.1104318, 0.1256006, 0.1378819, 0.1479658, 0.1551398
    0.1585819, 0.1574698, 0.1509815, 0.1385689, -0.2429053, -0.1787468, -0.1061024, -0.0281168
    0.0518019, 0.1301525, 0.2034337, 0.2681440, 0.3208122, 0.3594779, 0.3843636, 0.3958622
    0.3943667, 0.3802700, 0.3541828, -0.1525204, -0.0920759, -0.0272454, 0.0385099, 0.1026023
    0.1627523, 0.2166809, 0.2621090, 0.2967821, 0.3196711, 0.3315179, 0.3332026, 0.3256053
    0.3096063, 0.2860561, 0.0150660, 0.0434107, 0.0627593, 0.0694978, 0.0670999, 0.0615434
    0.0588093, 0.0648784, 0.0856273, 0.1217073, 0.1662185, 0.2116716, 0.2505772, 0.2754458
    0.2798735, 0.2162366, 0.2183650, 0.2233848, 0.2324456, 0.2441021, 0.2559917, 0.2657510
    0.2710166, 0.2694450, 0.2597000, 0.2419004, 0.2162787, 0.1830673, 0.1424989, 0.0952562
    0.1362316, 0.1365740, 0.1365937, 0.1362781, 0.1364811, 0.1383628, 0.1430836, 0.1518041
    0.1656370, 0.1833097, 0.2001021, 0.2110251, 0.2110893, 0.1953057, 0.1597695, 0.2693526
    0.2526301, 0.2290427, 0.1993189, 0.1654603, 0.1299180, 0.0951440, 0.0635899, 0.0376839
    0.0186739, 0.0061017, -0.0006241, -0.0020949, 0.0010980, 0.0083675, 0.0718948, 0.0736279
    0.0663077, 0.0486462, 0.0241959, -0.0017804, -0.0240178, -0.0372517, -0.0362922, -0.0197140
    0.0084689, 0.0438176, 0.0818932, 0.1182571, 0.1489090, 0.2040311, 0.1760602, 0.1488655
    0.1259609, 0.1088533, 0.0983406, 0.0952196, 0.1002875, 0.1143204, 0.1370499, 0.1666983
    0.2013704, 0.2391704, 0.2782030, 0.3165163, -0.0689507, -0.0382010, -0.0027471, 0.0360901
    0.0768460, 0.1180051, 0.1580521, 0.1954716, 0.2287414, 0.2560087, 0.2749425, 0.2831746
    0.2783364, 0.2580598, 0.2208492, 0.1579000, 0.1815706, 0.2018018, 0.2172008, 0.2264580
    0.2282930, 0.2214255, 0.2045750, 0.1764902, 0.1373646, 0.0894802, 0.0352822, -0.0227843
    -0.0822744, -0.1407132, 0.3488738, 0.3127563, 0.2706525, 0.2221488, 0.1696014, 0.1163450
    0.0657154, 0.0210487, -0.0143502, -0.0387152, -0.0525047, -0.0563509, -0.0508859, -0.0367417
    -0.0148446, 0.3615173, 0.3387830, 0.3187286, 0.3051912, 0.2983496, 0.2970895, 0.3002954
    0.3068514, 0.3156279, 0.3247805, 0.3314330, 0.3326287, 0.3254105, 0.3068217, 0.2747897
    0.0096716, 0.0130545, 0.0205799, 0.0341953, 0.0517230, 0.0695275, 0.0839715, 0.0914179
    0.0883023, 0.0747097, 0.0559986, 0.0379393, 0.0263023, 0.0268577, 0.0441777, 0.2673852
    0.2312898, 0.1902080, 0.1457800, 0.1007366, 0.0581942, 0.0212695, -0.0069210, -0.0233085
    -0.0272218, -0.0214552, -0.0090733, 0.0068592, 0.0232775, 0.0374092, 0.3126172, 0.3351676
    0.3537389, 0.3673866, 0.3753430, 0.3769028, 0.3713603, 0.3580105, 0.3361760, 0.3065886
    0.2720160, 0.2353852, 0.1996229, 0.1676558, 0.1419787, -0.0654669, -0.0718867, -0.0699960
    -0.0582158, -0.0376525, -0.0103616, 0.0216006, 0.0561774, 0.0913127, 0.1249676, 0.1551280
    0.1797818, 0.1969168, 0.2045209, 0.2011276, 0.0035095, 0.0267237, 0.0595774, 0.1021232
    0.1505744, 0.1997878, 0.2446186, 0.2799220, 0.3006223, 0.3050977, 0.2967178, 0.2792421
    0.2564301, 0.2320414, 0.2093303, 0.4031680, 0.3782132, 0.3430737, 0.2969676, 0.2423998
    0.1830370, 0.1225470, 0.0645977, 0.0128336, -0.0302647, -0.0638988, -0.0874017, -0.1001064
    -0.1013458, -0.0908780, -0.3787070, -0.3344548, -0.2683688, -0.1810184, -0.0790349, 0.0288080
    0.1337345, 0.2269686, 0.2998263, 0.3482294, 0.3747555, 0.3825019, 0.3745658, 0.3540447
    0.3239641, 0.1021986, 0.0784706, 0.0594509, 0.0483692, 0.0451714, 0.0486432, 0.0575691
    0.0707336, 0.0869172, 0.1047077, 0.1224141, 0.1383236, 0.1507237, 0.1579016, 0.1583659
    0.3241664, 0.2996249, 0.2704181, 0.2358454, 0.1967204, 0.1543916, 0.1102080, 0.0655189
    0.0216694, -0.0201885, -0.0591823, -0.0944615, -0.1251753, -0.1504731, -0.1695549, 0.2544329
    0.2891697, 0.3156454, 0.3320827, 0.3377355, 0.3322215, 0.3151588, 0.2861657, 0.2449083
    0.1934461, 0.1372975, 0.0822514, 0.0340964, -0.0013789, -0.0194179, 0.2888151, 0.2379840
    0.1856204, 0.1346230, 0.0870957, 0.0448620, 0.0097450, -0.0164324, -0.0318874, -0.0368578
    -0.0345013, -0.0282034, -0.0213498, -0.0173262, -0.0189599, 0.2968079, 0.2473975, 0.1997803
    0.1555224, 0.1146003, 0.0764289, 0.0404224, 0.0059948, -0.0274280, -0.0598468, -0.0904330
    -0.1182935, -0.1425350, -0.1622643, -0.1766483, -0.0011233, -0.0493377, -0.0840262, -0.1010937
    -0.1024579, -0.0921611, -0.0742478, -0.0527628, -0.0317155, -0.0133468, 0.0026578, 0.0168123
    0.0296309, 0.0416276, 0.0532006, 0.1971116, 0.1470363, 0.1037982, 0.0700926, 0.0455531
    0.0287313, 0.0181779, 0.0124431, 0.0100947, 0.0105579, 0.0144970, 0.0226735, 0.0358484
    0.0547832, 0.0797841, 0.3224356, 0.2951047, 0.2679510, 0.2422960, 0.2180237, 0.1945100
    0.1711301, 0.1472593, 0.1222822, 0.0960412, 0.0690413, 0.0418392, 0.0149912, -0.0109459
    -0.0353477, -0.1530922, -0.0787535, -0.0061018, 0.0639659, 0.1308371, 0.1939995, 0.2529409
    0.3071492, 0.3560962, 0.3984483, 0.4317082, 0.4532877, 0.4605985, 0.4510526, 0.4228450
    0.4657011, 0.4577034, 0.4349120, 0.3969806, 0.3471438, 0.2899017, 0.2297557, 0.1712074
    0.1186969, 0.0736097, 0.0329153, -0.0067610, -0.0487943, -0.0965596, -0.1523884, 0.2442393
    0.2262819, 0.2140083, 0.2105119, 0.2123847, 0.2139220, 0.2094161, 0.1931594, 0.1595427
    0.1078780, 0.0445891, -0.0233447, -0.0889442, -0.1452302, -0.1860809, 0.3310206, 0.3128510
    0.2919640, 0.2701569, 0.2472287, 0.2222723, 0.1943796, 0.1626428, 0.1261719, 0.0849796
    0.0403830, -0.0061989, -0.0533470, -0.0996426, -0.1435356, -0.0449725, -0.0561636, -0.0670867
    -0.0777271, -0.0852503, -0.0858250, -0.0756189, -0.0507998, -0.0076348, 0.0526256, 0.1215297
    0.1900634, 0.2492125, 0.2899631, 0.3048204, -0.0539522, -0.0477241, -0.0346324, -0.0135040
    0.0139166, 0.0448544, 0.0765331, 0.1061762, 0.1310467, 0.1503652, 0.1661818, 0.1807677
    0.1963939, 0.2153314, 0.2393548, -0.1637233, -0.1357918, -0.0938179, -0.0376610, 0.0279452
    0.0965447, 0.1616797, 0.2168922, 0.2558051, 0.2760912, 0.2812755, 0.2753401, 0.2622670
    0.2460382, 0.2300325, 0.0194602, 0.0524972, 0.0813316, 0.1019640, 0.1151623, 0.1233779
    0.1290647, 0.1346762, 0.1426255, 0.1532963, 0.1641391, 0.1723756, 0.1752274, 0.1699161
    0.1542903, -0.0220697, -0.0453485, -0.0583201, -0.0572203, -0.0436282, -0.0210112, 0.0071615
    0.0374204, 0.0663070, 0.0909032, 0.1090723, 0.1187383, 0.1178255, 0.1042580, 0.0766757
    0.3994047, 0.4100869, 0.4076762, 0.3903410, 0.3592589, 0.3166709, 0.2648189, 0.2059451
    0.1422955, 0.0763156, 0.0107389, -0.0516787, -0.1081810, -0.1560123, -0.1927040, 0.0080644
    0.0036825, 0.0026532, 0.0063896, 0.0139113, 0.0233915, 0.0330028, 0.0409177, 0.0453350
    0.0457655, 0.0436165, 0.0404436, 0.0378019, 0.0372470, 0.0400603, 0.0514523, 0.0645745
    0.0733467, 0.0745991, 0.0700726, 0.0632432, 0.0575892, 0.0565885, 0.0636614, 0.0793326
    0.0999418, 0.1215024, 0.1400274, 0.1515301, 0.1526694, -0.1089400, -0.0601436, -0.0094093
    0.0410700, 0.0888106, 0.1312256, 0.1657280, 0.1897310, 0.2006824, 0.1977701, 0.1826966
    0.1573610, 0.1236620, 0.0834987, 0.0389159, -0.2293558, -0.2457530, -0.2540689, -0.2519087
    -0.2395357, -0.2181525, -0.1889627, -0.1531701, -0.1119761, -0.0664704, -0.0175811, 0.0337764
    0.0866864, 0.1402335, 0.1932246, -0.0014453, 0.0427826, 0.0782020, 0.1006542, 0.1101948
    0.1083684, 0.0967214, 0.0768001, 0.0501726, 0.0194903, -0.0110291, -0.0370458, -0.0542200
    -0.0582117, -0.0456701, 0.1513067, 0.1696866, 0.1851027, 0.1943745, 0.1975931, 0.1960054
    0.1908595, 0.1834036, 0.1748806, 0.1662717, 0.1581791, 0.1511759, 0.1458349, 0.1427290
    0.1422020, -0.2066851, -0.1963823, -0.1819667, -0.1621342, -0.1364758, -0.1048992, -0.0673125
    -0.0236236, 0.0262254, 0.0805904, 0.1353675, 0.1862607, 0.2289738, 0.2592110, 0.2733612
    -0.0941582, -0.0843463, -0.0741668, -0.0629804, -0.0504810, -0.0364804, -0.0207905, -0.0032232
    0.0164070, 0.0381581, 0.0619032, 0.0875013, 0.1148112, 0.1436917, 0.1737317, 0.2887293
    0.2803732, 0.2718796, 0.2641100, 0.2556263, 0.2441782, 0.2275138, 0.2033819, 0.1695814
    0.1264466, 0.0779753, 0.0284514, -0.0178413, -0.0566190, -0.0841949, 0.3184404, 0.2659197
    0.2130646, 0.1655213, 0.1247574, 0.0907645, 0.0635325, 0.0430512, 0.0292952, 0.0214715
    0.0176783, 0.0159269, 0.0142289, 0.0105958, 0.0034388, -0.0530774, -0.0185990, 0.0176381
    0.0541214, 0.0901813, 0.1254463, 0.1595450, 0.1921062, 0.2227451, 0.2503918, 0.2729866
    0.2883926, 0.2944729, 0.2890907, 0.2706394, 0.0241861, 0.0194550, 0.0078640, -0.0127113
    -0.0401709, -0.0709218, -0.1013695, -0.1279195, -0.1470182, -0.1571724, -0.1598653, -0.1568129
    -0.1497310, -0.1403356, -0.1301921, -0.2220779, -0.1384692, -0.0615650, 0.0008017, 0.0490883
    0.0866810, 0.1169699, 0.1433445, 0.1691667, 0.1963915, 0.2249406, 0.2545775, 0.2850651
    0.3161669, 0.3472719, -0.1260286, -0.0687067, -0.0169450, 0.0260598, 0.0603338, 0.0870414
    0.1073486, 0.1224212, 0.1334223, 0.1413819, 0.1471374, 0.1515112, 0.1553256, 0.1594029
    0.1643221, 0.0679620, 0.0569232, 0.0502098, 0.0525103, 0.0620255, 0.0746641, 0.0863320
    0.0929350, 0.0904486, 0.0783332, 0.0610852, 0.0435940, 0.0307494, 0.0274407, 0.0375336
    0.2703077, 0.2632689, 0.2419729, 0.2056639, 0.1574999, 0.1020222, 0.0437732, -0.0127044
    -0.0629007, -0.1039434, -0.1353271, -0.1567311, -0.1678347, -0.1683172, -0.1582271, 0.0847183
    0.1098696, 0.1312823, 0.1483144, 0.1606050, 0.1678921, 0.1699141, 0.1664094, 0.1571405
    0.1430880, 0.1269924, 0.1117319, 0.1001844, 0.0952279, 0.0990615, 0.0977777, 0.0974152
    0.1030202, 0.1133846, 0.1268590, 0.1416382, 0.1559168, 0.1678891, 0.1757804, 0.1793439
    0.1805413, 0.1815066, 0.1843741, 0.1912779, 0.2037512, 0.1948271, 0.1585226, 0.1284160
    0.1096051, 0.1004121, 0.0967657, 0.0945914, 0.0898151, 0.0784211, 0.0593341, 0.0357279
    0.0111078, -0.0110205, -0.0271515, -0.0343787, -0.0583804, -0.0492346, -0.0246846, 0.0179968
    0.0750689, 0.1405060, 0.2082794, 0.2723607, 0.3267582, 0.3673198, 0.3925519, 0.4011690
    0.3918851, 0.3634143, 0.3153024, -0.0799121, -0.0382486, 0.0174844, 0.0900423, 0.1732106
    0.2576053, 0.3338386, 0.3925231, 0.4243912, 0.4261967, 0.4033940, 0.3621175, 0.3085012
    0.2486794, 0.1883862, -0.0054998, 0.0268777, 0.0642457, 0.1062926, 0.1500708, 0.1917013
    0.2273039, 0.2529988, 0.2649571, 0.2619151, 0.2463168, 0.2208953, 0.1883839, 0.1515156
    0.1129520, 0.0002639, -0.0171350, -0.0190994, -0.0002053, 0.0366840, 0.0857773, 0.1412798
    0.1973969, 0.2483612, 0.2897698, 0.3191915, 0.3343496, 0.3329667, 0.3127661, 0.2725430
    0.1266231, 0.1203523, 0.1191382, 0.1251075, 0.1365440, 0.1503732, 0.1635192, 0.1729061
    0.1754818, 0.1693808, 0.1544532, 0.1306830, 0.0980539, 0.0565500, 0.0066180, 0.3656715
    0.3636282, 0.3567902, 0.3451262, 0.3302327, 0.3142814, 0.2994444, 0.2878943, 0.2817798
    0.2820802, 0.2880843, 0.2989489, 0.3138308, 0.3318869, 0.3522008, 0.2191025, 0.2088497
    0.1824610, 0.1379277, 0.0805443, 0.0181859, -0.0412694, -0.0899436, -0.1200651, -0.1291905
    -0.1225768, -0.1060824, -0.0855652, -0.0668837, -0.0551411, 0.2840573, 0.2606719, 0.2421650
    0.2330887, 0.2319341, 0.2350508, 0.2387860, 0.2394869, 0.2335495, 0.2198247, 0.2007100
    0.1788805, 0.1570106, 0.1377753, 0.1234751, -0.0127013, 0.0015273, 0.0183003, 0.0372849
    0.0590537, 0.0844991, 0.1145137, 0.1499904, 0.1917651, 0.2378330, 0.2820836, 0.3180861
    0.3394094, 0.3396227, 0.3136386, 0.3303948, 0.2962694, 0.2639709, 0.2383179, 0.2185149
    0.2017822, 0.1853379, 0.1664001, 0.1422200, 0.1117032, 0.0761464, 0.0370327, -0.0041545
    -0.0459320, -0.0868411, 0.4776590, 0.4405926, 0.3831118, 0.3045344, 0.2117887, 0.1144919
    0.0222643, -0.0552737, -0.1086263, -0.1345284, -0.1387190, -0.1276404, -0.1077348, -0.0854444
    -0.0665031, 0.2472814, 0.2532029, 0.2554891, 0.2537187, 0.2481505, 0.2392831, 0.2276159
    0.2136479, 0.1978746, 0.1806120, 0.1619159, 0.1418223, 0.1203668, 0.0975853, 0.0736581
    0.2909483, 0.2541333, 0.2200389, 0.1913712, 0.1664122, 0.1418806, 0.1144933, 0.0809673
    0.0380919, -0.0137120, -0.0687756, -0.1210205, -0.1643681, -0.1927401, -0.2011514, 0.3269688
    0.2871901, 0.2487628, 0.2146654, 0.1840793, 0.1548441, 0.1247982, 0.0917795, 0.0536782
    0.0109738, -0.0321111, -0.0710617, -0.1013634, -0.1185014, -0.1188881, 0.0946175, 0.0890556
    0.0793130, 0.0646631, 0.0476779, 0.0320955, 0.0216552, 0.0200963, 0.0310874, 0.0547607
    0.0861372, 0.1198392, 0.1504888, 0.1727082, 0.1819699, 0.0393857, 0.0173748, 0.0074503
    0.0122309, 0.0284274, 0.0506631, 0.0735588, 0.0917353, 0.0998738, 0.0956635, 0.0811420
    0.0586859, 0.0306720, -0.0005228, -0.0325484, 0.0451037, 0.0401532, 0.0413506, 0.0486539
    0.0615390, 0.0793113, 0.1012761, 0.1267387, 0.1549934, 0.1847907, 0.2140950, 0.2408091
    0.2628361, 0.2780790, 0.2846137, 0.4447103, 0.4606536, 0.4620782, 0.4464465, 0.4154837
    0.3724217, 0.3204935, 0.2629325, 0.2029840, 0.1444890, 0.0921497, 0.0507353, 0.0250152
    0.0197588, 0.0383635, 0.0113983, -0.0025411, -0.0095421, -0.0090760, -0.0001719, 0.0182980
    0.0474615, 0.0884463, 0.1422959, 0.2058322, 0.2697761, 0.3243722, 0.3598652, 0.3664997
    0.3366227, 0.4379125, 0.4340893, 0.4142609, 0.3746997, 0.3180538, 0.2492237, 0.1731127
    0.0946240, 0.0186531, -0.0502976, -0.1082933, -0.1514438, -0.1758586, -0.1776474, -0.1538772
    0.0435713, 0.1023890, 0.1571982, 0.2042765, 0.2428561, 0.2732129, 0.2956241, 0.3103669
    0.3177248, 0.3182969, 0.3131383, 0.3033400, 0.2899927, 0.2741874, 0.2569061, -0.0169530
    0.0482630, 0.1006642, 0.1347321, 0.1525192, 0.1587533, 0.1581649, 0.1554849, 0.1553766
    0.1591473, 0.1632528, 0.1637703, 0.1567772, 0.1383508, 0.1055693, 0.1640725, 0.2193762
    0.2633009, 0.2910420, 0.3032644, 0.3025660, 0.2915466, 0.2728062, 0.2489394, 0.2222756
    0.1947605, 0.1683103, 0.1448407, 0.1262679, 0.1141124, 0.3087527, 0.2934167, 0.2687906
    0.2355407, 0.1968128, 0.1566285, 0.1190106, 0.0879818, 0.0675041, 0.0585042, 0.0575218
    0.0607541, 0.0643983, 0.0646518, 0.0583238, -0.1016200, -0.1381792, -0.1526069, -0.1422335
    -0.1110120, -0.0652358, -0.0112011, 0.0447964, 0.0965116, 0.1402643, 0.1760802, 0.2042744
    0.2251620, 0.2390581, 0.2462893, 0.1279266, 0.1642068, 0.2040457, 0.2468100, 0.2889968
    0.3260885, 0.3535664, 0.3669118, 0.3616712, 0.3366445, 0.2953336, 0.2416076, 0.1793356
    0.1123866, 0.0446456, 0.1672688, 0.1691973, 0.1596964, 0.1362852, 0.1028221, 0.0654058
    0.0301374, 0.0031179, -0.0096328, -0.0061744, 0.0095387, 0.0330917, 0.0600698, 0.0860583
    0.1070712, -0.0964169, -0.0313356, 0.0260206, 0.0718114, 0.1082190, 0.1395537, 0.1701279
    0.2042545, 0.2461682, 0.2962097, 0.3490918, 0.3990881, 0.4404719, 0.4675168, 0.4753764
    -0.0489389, -0.0850012, -0.1125917, -0.1296344, -0.1367418, -0.1354762, -0.1274011, -0.1140797
    -0.0970774, -0.0780595, -0.0588351, -0.0412249, -0.0270492, -0.0181288, -0.0158684, 0.1477952
    0.1688908, 0.1754669, 0.1630533, 0.1347361, 0.0962714, 0.0534185, 0.0119364, -0.0224687
    -0.0467487, -0.0616961, -0.0684036, -0.0679637, -0.0614692, -0.0500232, 0.1645879, 0.1614200
    0.1560836, 0.1482218, 0.1372024, 0.1222956, 0.1027718, 0.0779012, 0.0469888, 0.0110787
    -0.0262715, -0.0613082, -0.0902775, -0.1094258, -0.1156644, 0.0850691, 0.0824022, 0.0861316
    0.0978422, 0.1145259, 0.1315515, 0.1442859, 0.1480960, 0.1384219, 0.1143626, 0.0803052
    0.0410497, 0.0013958, -0.0338564, -0.0604551, 0.0698737, 0.0935514, 0.1118281, 0.1234716
    0.1297737, 0.1329181, 0.1350895, 0.1384727, 0.1452090, 0.1552661, 0.1654707, 0.1724038
    0.1726468, 0.1627811, 0.1402190, 0.2121026, 0.1936445, 0.1779399, 0.1671628, 0.1613881
    0.1599490, 0.1621778, 0.1674068, 0.1749513, 0.1832833, 0.1896554, 0.1912252, 0.1851500
    0.1685875, 0.1395548, 0.2552460, 0.2744880, 0.2878085, 0.2938685, 0.2918869, 0.2812796
    0.2614624, 0.2318516, 0.1918945, 0.1426111, 0.0872940, 0.0294130, -0.0275617, -0.0801603
    -0.1251423, 0.0897723, 0.1295542, 0.1695995, 0.2061170, 0.2365225, 0.2586586, 0.2703682
    0.2694940, 0.2539237, 0.2237770, 0.1823998, 0.1333898, 0.0803446, 0.0268620, -0.0237097
    -0.0012536, -0.0044433, 0.0036227, 0.0243809, 0.0565675, 0.0979643, 0.1463522, 0.1995119
    0.2552006, 0.3099911, 0.3587447, 0.3961890, 0.4170515, 0.4160601, 0.3891635, 0.1413942
    0.0918267, 0.0525317, 0.0284236, 0.0203599, 0.0277650, 0.0500616, 0.0866723, 0.1369660
    0.1976304, 0.2614771, 0.3210156, 0.3687549, 0.3972047, 0.4001647, 0.0071008, 0.0141330
    0.0175140, 0.0171941, 0.0140665, 0.0093580, 0.0042957, 0.0001066, -0.0019958, -0.0014767
    0.0012181, 0.0055659, 0.0110443, 0.0171307, 0.0232980, 0.1677007, 0.1440248, 0.1260456
    0.1154603, 0.1106566, 0.1088534, 0.1072679, 0.1031174, 0.0936591, 0.0781428, 0.0586985
    0.0376811, 0.0174452, 0.0003458, -0.0116552, 0.2191785, 0.1754734, 0.1363627, 0.1054419
    0.0809361, 0.0591724, 0.0364760, 0.0091720, -0.0263512, -0.0705335, -0.1192316, -0.1679444
    -0.2121706, -0.2474090, -0.2697828, 0.0425201, 0.0156578, 0.0015893, 0.0034433, 0.0182595
    0.0409261, 0.0663287, 0.0893530, 0.1049407, 0.1108327, 0.1088154, 0.1009912, 0.0894624
    0.0763314, 0.0634977, -0.1136051, -0.1340698, -0.1425093, -0.1343604, -0.1120891, -0.0806456
    -0.0449827, -0.0100533, 0.0192500, 0.0410470, 0.0578115, 0.0723571, 0.0874974, 0.1060461
    0.1301388, 0.3223215, 0.2939837, 0.2588057, 0.2166909, 0.1685311, 0.1155670, 0.0590401
    0.0001918, -0.0597306, -0.1191781, -0.1761660, -0.2286753, -0.2746871, -0.3121828, -0.3393981
    -0.0935562, -0.1333105, -0.1554120, -0.1551125, -0.1358413, -0.1039169, -0.0656612, -0.0273958
    0.0046289, 0.0277544, 0.0445121, 0.0578388, 0.0706711, 0.0859459, 0.1058997, -0.2922828
    -0.3223130, -0.3397177, -0.3384411, -0.3181745, -0.2806396, -0.2275603, -0.1606608, -0.0816946
    0.0061060, 0.0973715, 0.1865656, 0.2681519, 0.3365944, 0.3869630, 0.2643729, 0.2746395
    0.2614893, 0.2177395, 0.1499089, 0.0693582, -0.0125465, -0.0844391, -0.1350913, -0.1601707
    -0.1653113, -0.1569250, -0.1414238, -0.1252196, -0.1138501, 0.4354936, 0.4341073, 0.4179850
    0.3832615, 0.3326827, 0.2713305, 0.2042893, 0.1366438, 0.0734248, 0.0169786, -0.0342286
    -0.0820333, -0.1282721, -0.1747817, -0.2229370, -0.1664707, -0.1421772, -0.1170454, -0.0914960
    -0.0632192, -0.0289405, 0.0146161, 0.0707263, 0.1425602, 0.2280037, 0.3173051, 0.4001171
    0.4660917, 0.5048816, 0.5080253, -0.1292062, -0.1389786, -0.1378920, -0.1246152, -0.1018512
    -0.0737288, -0.0443782, -0.0179297, 0.0015483, 0.0130853, 0.0201883, 0.0267135, 0.0365173
    0.0534560, 0.0804509, -0.0730679, -0.0154378, 0.0334601, 0.0697915, 0.0953205, 0.1137892
    0.1289420, 0.1445232, 0.1642243, 0.1890954, 0.2163684, 0.2429774, 0.2658562, 0.2819392
    0.2885647, 0.0196449, 0.1075124, 0.1749331, 0.2112231, 0.2192439, 0.2066427, 0.1810724
    0.1501857, 0.1215775, 0.0999386, 0.0857626, 0.0792158, 0.0804643, 0.0896742, 0.1065843
    -0.0294458, -0.0252217, -0.0179748, -0.0076381, 0.0057341, 0.0220445, 0.0411958, 0.0630908
    0.0876141, 0.1137514, 0.1391886, 0.1615103, 0.1783011, 0.1871457, 0.1860997, -0.1970514
    -0.1357522, -0.0762910, -0.0224621, 0.0250597, 0.0667014, 0.1028913, 0.1340579, 0.1606202
    0.1825256, 0.1990407, 0.2093787, 0.2127527, 0.2083761, 0.1957602, -0.0285414, 0.0054047
    0.0385091, 0.0682716, 0.0945044, 0.1178371, 0.1389001, 0.1583238, 0.1767277, 0.1941800
    0.2099522, 0.2232538, 0.2332940, 0.2392823, 0.2405044, 0.0658678, 0.0158323, -0.0245650
    -0.0521899, -0.0660890, -0.0660789, -0.0519775, -0.0236025, 0.0191778, 0.0739659, 0.1347086
    0.1950676, 0.2487045, 0.2892808, 0.3113863, -0.0085855, -0.0287831, -0.0534990, -0.0824288
    -0.1123461, -0.1389922, -0.1581070, -0.1654305, -0.1567752, -0.1315818, -0.0945342, -0.0507258
    -0.0052501, 0.0367995, 0.0709051, 0.0738313, 0.0684976, 0.0679310, 0.0731166, 0.0834564
    0.0977930, 0.1149683, 0.1338241, 0.1532058, 0.1721224, 0.1898203, 0.2055642, 0.2186189
    0.2282491, 0.2338492, 0.1159662, 0.1395010, 0.1531870, 0.1542170, 0.1446029, 0.1280593
    0.1083025, 0.0890493, 0.0739853, 0.0652543, 0.0627720, 0.0662800, 0.0755200, 0.0902336
    0.1099432, 0.1603437, 0.1409672, 0.1301730, 0.1314190, 0.1422498, 0.1581202, 0.1744828
    0.1867900, 0.1905443, 0.1837432, 0.1679905, 0.1451715, 0.1171716, 0.0858760, 0.0531268
    -0.0067003, 0.0422367, 0.0862258, 0.1194893, 0.1407797, 0.1504502, 0.1488556, 0.1363510
    0.1133452, 0.0829410, 0.0521345, 0.0282259, 0.0185155, 0.0303034, 0.0692947, -0.1397834
    -0.1226367, -0.0998779, -0.0727695, -0.0440968, -0.0171836, 0.0046458, 0.0180672, 0.0198232
    0.0100043, -0.0064608, -0.0242657, -0.0381036, -0.0426683, -0.0338483, -0.0392564, -0.0623119
    -0.0796157, -0.0887345, -0.0888502, -0.0797154, -0.0610837, -0.0327086, 0.0056304, 0.0528399
    0.1059276, 0.1617535, 0.2171771, 0.2690582, 0.3144290, -0.0844851, -0.1169414, -0.1316300
    -0.1229434, -0.0945529, -0.0534092, -0.0064662, 0.0393218, 0.0770692, 0.1033218, 0.1195838
    0.1277469, 0.1297024, 0.1273420, 0.1224143, -0.0281096, -0.0492643, -0.0617397, -0.0620934
    -0.0524887, -0.0370700, -0.0199838, -0.0053767, 0.0026565, 0.0026123, -0.0032682, -0.0124515
    -0.0224041, -0.0305924, -0.0347535, 0.1162144, 0.1162464, 0.1152539, 0.1149707, 0.1160708
    0.1188535, 0.1236179, 0.1306628, 0.1402802, 0.1524059, 0.1664614, 0.1818278, 0.1978863
    0.2140184, 0.2294946, -0.3531238, -0.3113537, -0.2564495, -0.1873008, -0.1075008, -0.0223050
    0.0630295, 0.1432453, 0.2131329, 0.2698757, 0.3141150, 0.3467622, 0.3687286, 0.3809256
    0.3842045, -0.1884619, -0.1628718, -0.1350373, -0.1068904, -0.0778529, -0.0464595, -0.0112437
    0.0292606, 0.0764759, 0.1296297, 0.1847768, 0.2377247, 0.2842804, 0.3202514, 0.3420023
    -0.1447252, -0.0873921, -0.0393342, -0.0056648, 0.0136374, 0.0204073, 0.0164821, 0.0036989
    -0.0161070, -0.0411906, -0.0699381, -0.1007457, -0.1320096, -0.1621261, -0.1895159, -0.0127307
    0.0115193, 0.0246389, 0.0227765, 0.0088583, -0.0117947, -0.0338587, -0.0520098, -0.0609936
    -0.0590198, -0.0493051, -0.0354570, -0.0210829, -0.0097904, -0.0046570, -0.2706166, -0.2152561
    -0.1614663, -0.1131052, -0.0710059, -0.0349327, -0.0046484, 0.0200838, 0.0394980, 0.0536839
    0.0625218, 0.0658757, 0.0636099, 0.0555885, 0.0418838, 0.1682657, 0.2014977, 0.2363719
    0.2719665, 0.3033067, 0.3239860, 0.3275956, 0.3077274, 0.2581241, 0.1801004, 0.0859136
    -0.0113247, -0.0985027, -0.1625091, -0.1924079, 0.1548493, 0.1274848, 0.0930780, 0.0527419
    0.0073450, -0.0423309, -0.0955039, -0.1513921, -0.2091717, -0.2659172, -0.3156655, -0.3522164
    -0.3693698, -0.3609255, -0.3222212, -0.2979792, -0.2424090, -0.1887240, -0.1413078, -0.0992972
    -0.0599756, -0.0206240, 0.0214765, 0.0689689, 0.1207091, 0.1700784, 0.2100313, 0.2335221
    0.2335050, 0.2046276, 0.0092246, 0.0359160, 0.0440331, 0.0295438, -0.0022919, -0.0429304
    -0.0838242, -0.1164263, -0.1322996, -0.1285388, -0.1102317, -0.0830908, -0.0528282, -0.0251560
    -0.0051098, -0.2077721, -0.1428818, -0.0750517, -0.0063251, 0.0604656, 0.1222094, 0.1757949
    0.2181106, 0.2460871, 0.2587606, 0.2582098, 0.2467509, 0.2267002, 0.2003741, 0.1699104
    0.1926296, 0.1996422, 0.1957717, 0.1782260, 0.1507380, 0.1193459, 0.0900907, 0.0690134
    0.0620527, 0.0700283, 0.0863623, 0.1038991, 0.1154830, 0.1139586, 0.0935857, 0.2540199
    0.2200293, 0.1836706, 0.1470135, 0.1120644, 0.0808076, 0.0552274, 0.0373081, 0.0289894
    0.0299858, 0.0367958, 0.0456668, 0.0528462, 0.0545814, 0.0477988, 0.2381483, 0.1698887
    0.1093040, 0.0629906, 0.0289852, 0.0023004, -0.0220547, -0.0490711, -0.0836546, -0.1264556
    -0.1719740, -0.2142296, -0.2472422, -0.2650316, -0.2627318, 0.1960691, 0.1902413, 0.1806788
    0.1657014, 0.1467573, 0.1264002, 0.1071849, 0.0916663, 0.0823652, 0.0800960, 0.0832075
    0.0898558, 0.0981969, 0.1063871, 0.1127269, 0.2066814, 0.1657172, 0.1147147, 0.0570145
    -0.0038562, -0.0643041, -0.1207360, -0.1695584, -0.2072266, -0.2326268, -0.2481574, -0.2564919
    -0.2603031, -0.2622641, -0.2645970, 0.3111595, 0.2355734, 0.1618845, 0.0949096, 0.0363203
    -0.0133232, -0.0534619, -0.0835368, -0.1030114, -0.1124611, -0.1140693, -0.1101447, -0.1029961
    -0.0949322, -0.0879785, 0.1739859, 0.1719795, 0.1621039, 0.1448733, 0.1223166, 0.0969976
    0.0714810, 0.0483313, 0.0300843, 0.0178369, 0.0106066, 0.0072484, 0.0066175, 0.0075690
    0.0090559, 0.4547790, 0.3999088, 0.3345425, 0.2604879, 0.1808922, 0.0993766, 0.0195626
    -0.0549284, -0.1205168, -0.1757313, -0.2221463, -0.2615746, -0.2958284, -0.3267205, -0.3555478];

   // MatMul 'l0_base': W(16×28) + b(16)
   w2 : ARRAY[0..463] OF REAL :=
[0.6531532, 1.1509302, 0.8542801, 0.1212990, 0.6904182, -0.5414373, -0.9088417, -0.5722627
    0.8944874, 0.5538955, -1.0278374, -0.4903141, -0.1389806, 0.4674363, -1.0210936, -0.6274210
    0.2741612, 1.0625501, -0.9149109, -0.7328060, 0.7575151, -0.2042419, -0.2723309, -0.7191657
    -0.0280776, 0.2011455, -0.3273573, -0.4418836, 1.2626092, 1.2265757, 1.5492810, -0.5662438
    -0.9511591, 0.1725382, 1.2004387, -0.0104933, 1.5757133, 1.6623878, 1.2453479, 0.1729178
    0.2919613, 0.0309749, -0.6492561, -0.3796145, -0.5120577, 0.3172240, -0.4038502, 0.5928957
    -0.5418487, -0.5144768, -0.7627655, 0.8234128, -0.4605753, -0.7895154, 0.0910844, -0.6752480
    0.0697802, -0.4284368, 0.0479970, 0.0784096, -0.0238369, 0.0168181, -0.8319796, 0.1763645
    0.2104895, 0.8926834, 0.6908084, 0.4001502, -0.3938401, 0.1085153, -0.6449838, -0.7566856
    -0.0827282, 0.4948159, -1.1559126, -0.5277553, 0.8248507, 0.1181727, 0.7966241, 0.2058670
    -0.8326430, -0.1626337, -0.0323979, -0.2344580, -1.5619131, -1.4697499, -1.8048265, -0.8762984
    -1.3497895, -0.8686097, -0.9026392, -0.7284883, -1.7362306, -0.0363061, 1.1192808, 0.8043320
    -0.1950512, -0.3716736, -0.4853409, -0.5649784, -0.4172391, 0.6161152, -0.6759697, 0.0904574
    0.5806844, 0.6348718, 0.7333751, 0.6839716, -0.3869329, 0.5344537, 0.9650685, 0.0383124
    -0.8913731, -0.3576556, -0.6536014, -0.0847967, -0.0349820, 0.5889089, -0.2677067, -0.2245978
    -0.5749647, -0.9168990, -0.6333076, -0.4074411, 0.4441338, 0.1501607, -0.1995225, 0.7596117
    0.0808029, -0.3484810, -0.0210259, 0.9137757, -0.7801852, -0.2238004, -0.3275166, -0.0392269
    -0.2500529, 0.1511434, -0.2167200, 0.2951781, 0.3186197, 0.0769461, 0.4348049, -0.2419707
    -0.3043656, -0.3270995, 0.5164679, 0.4538959, 0.2316195, 0.8929619, 1.3953813, 0.6482492
    -0.2139386, -0.0555586, -0.2996079, -0.7336348, -0.7894226, 0.6769296, -1.0865229, 0.9084685
    0.4970312, 0.3730805, 0.6737831, 0.5160832, -0.8191277, 0.0919100, 0.4878978, -0.4577431
    0.5415249, 0.0459770, 0.2380498, 0.3544105, 0.0758338, 0.5700713, -0.3280728, 0.0073880
    0.9576581, -0.1927161, -0.5408630, 0.3759742, -0.3697540, -0.4095958, 0.2953050, -0.3224963
    0.4659955, 0.2666524, 0.7817978, -0.3882965, 0.5259117, 0.1157550, -0.0868794, 0.1442592
    0.4463586, -0.0788809, 0.3359323, 0.3131578, -0.2152938, 0.8472598, 0.6115276, -0.3911876
    0.0704370, -0.2515413, 0.8549601, 0.3596184, -0.5991781, -1.2437032, -0.1800027, -1.1388100
    0.5647227, 0.3254773, -0.8980638, 0.6457720, 0.9825901, -0.7528893, 0.0748151, 0.1365464
    -0.6619212, -0.1892451, -0.3664528, -0.7725444, -0.1610090, -0.1782233, -0.1539104, -0.0613308
    1.0186411, -0.0857887, -0.3516517, 0.3065239, 0.0238268, 0.2399618, -0.2922754, -0.1875871
    1.1885412, -0.1608811, -1.1761448, -0.3997688, -1.0060421, 0.0516912, 0.4627137, -1.1369811
    0.6643242, 0.2780860, 0.0209994, -0.6893836, 0.5776726, -0.0303992, -0.2795104, -0.2218146
    0.4949092, 0.1933563, -0.3510525, 0.0224845, -1.5212339, -1.1815313, -1.4145346, 0.4340951
    0.3062091, 0.0455918, -0.3191082, 0.2872083, -1.7960831, -0.9681343, -0.2131347, -0.0914112
    0.4054331, -0.9982103, -0.5022178, 0.3359171, 0.8721167, -0.0940284, -1.9242376, 0.1256431
    -0.4745836, 0.5358467, 0.1780284, -0.2262570, -0.6270480, -0.4930463, -0.6283804, 0.2633540
    0.2300479, 1.1844879, 0.6107946, -0.2428536, 0.4828842, 0.1695227, 0.5681323, 0.2884444
    0.2841129, -0.8758434, 0.2491129, -0.3859273, -0.4150312, 0.4644483, 0.1481924, -0.4265237
    0.3190451, -0.6888376, 0.8258311, 0.4234703, 0.0811714, -0.2619098, -1.0289083, -0.8263102
    0.5947338, -0.0104262, 0.4936709, 0.0368680, 0.0356015, 0.8885249, 0.5964210, -0.0492413
    -0.1171272, -0.2020979, 0.5844330, -0.0603527, -0.1831383, -1.3109881, -0.5292199, 0.0204109
    0.2865884, -0.0319725, -0.1081036, 0.6079996, 0.7452201, -0.9360539, 0.2803982, 0.5940919
    -0.3924443, -0.0010045, -0.2540028, -0.1956804, 0.3307257, -0.0851964, 0.0121359, 0.2464700
    -1.3067886, -1.2725198, -1.4913075, 0.6236749, 0.3114894, 0.3706363, -0.5315891, 0.3905119
    -1.4648223, -0.4327554, -0.1879684, -0.2010098, 0.5315167, -0.0843144, 0.0634309, 0.3992346
    0.3824810, -0.0483803, -0.2913157, 0.0982564, -0.4671767, 0.1136492, 0.0548117, -0.2728889
    -0.4076180, -0.4225101, -0.2261286, 0.2782121, 0.7695327, 0.2566034, 0.1953621, 0.0408440
    0.0124786, 0.2488524, -0.5697264, 0.0825308, 0.8317476, -0.8402474, -1.0685767, -0.2165811
    -0.4149429, -0.3753743, 0.1834853, 0.0865243, 0.7913322, -0.3387795, 0.5137359, -0.3165046
    0.2458227, 0.3609711, -0.3399727, -0.8827292, 0.4816631, 0.3397982, 0.1536530, 0.1695612
    0.5854009, -0.0813269, 0.1311246, 0.0674454, 0.2877986, -0.2290608, -0.6208226, -0.5486314
    0.9404889, 0.4580346, -0.5092251, -0.5765274, -0.4888373, 0.0444687, -0.2916232, -0.8206158
    0.2447187, 0.4721361, -0.6585346, -0.6879834, 0.5628800, 0.0532022, 0.1965619, 0.0561261
    0.2354458, 0.3610592, 0.0144084, 0.1184748, 0.0501975, 0.1787246, 0.4878071, 0.1703812
    0.1714815, -0.0600145, 0.7518312, 0.4750999, -0.1374112, 1.2641517, 1.2422327, 0.3578296
    -0.3659381, 0.3438349, -0.3962274, -0.3011864, -0.1204108, 0.3932763, -0.0552154, 0.3200105
    0.7434683, 0.4552981, 0.4342712, 0.2647173, -0.2187249, -0.2678579, 0.1962206, -0.4789418
    0.0, 0.0, 0.0, 0.0, 0.0, 0.0, 0.0, 0.0
    0.0, 0.0, 0.0, 0.0, 0.0, 0.0, 0.0, 0.0];

   // BsplineLUT 'l1_bspline': grid(15 pts) + table(4×16×15)
   w3 : ARRAY[0..14] OF REAL :=
[-3.0000000, -2.5714286, -2.1428571, -1.7142857, -1.2857143, -0.8571429, -0.4285714, 0.0
    0.4285714, 0.8571429, 1.2857143, 1.7142857, 2.1428571, 2.5714286, 3.0000000];
   w4 : ARRAY[0..959] OF REAL :=
[0.1180185, 0.1203233, 0.1224589, 0.1244152, 0.1261825, 0.1277508, 0.1291103, 0.1302511
    0.1311632, 0.1318369, 0.1322627, 0.1324407, 0.1323814, 0.1320955, 0.1315938, 0.0842773
    0.0825064, 0.0806832, 0.0787976, 0.0768397, 0.0747991, 0.0726658, 0.0704296, 0.0680806
    0.0656084, 0.0630035, 0.0602665, 0.0574086, 0.0544416, 0.0513772, 0.0936770, 0.0899939
    0.0863021, 0.0826108, 0.0789293, 0.0752668, 0.0716325, 0.0680359, 0.0644860, 0.0609922
    0.0575636, 0.0542039, 0.0509117, 0.0476852, 0.0445227, 0.0226024, 0.0203358, 0.0180222
    0.0156702, 0.0132885, 0.0108859, 0.0084710, 0.0060526, 0.0036394, 0.0012401, -0.0011365
    -0.0034818, -0.0057870, -0.0080435, -0.0102426, -0.0585543, -0.0502811, -0.0417866, -0.0330670
    -0.0241186, -0.0149379, -0.0055211, 0.0041354, 0.0140353, 0.0241822, 0.0345793, 0.0452160
    0.0560676, 0.0671089, 0.0783146, 0.0506554, 0.0470260, 0.0433342, 0.0395754, 0.0357449
    0.0318381, 0.0278503, 0.0237768, 0.0196131, 0.0153543, 0.0109963, 0.0065434, 0.0020089
    -0.0025934, -0.0072500, 0.0495298, 0.0382326, 0.0269749, 0.0157830, 0.0046829, -0.0062993
    -0.0171372, -0.0278048, -0.0382758, -0.0485243, -0.0585243, -0.0682607, -0.0777291, -0.0869256
    -0.0958461, 0.0110217, 0.0143777, 0.0176291, 0.0207730, 0.0238068, 0.0267275, 0.0295325
    0.0322190, 0.0347841, 0.0372252, 0.0395394, 0.0417255, 0.0437835, 0.0457136, 0.0475160
    0.1000672, 0.0975504, 0.0949741, 0.0923415, 0.0896557, 0.0869198, 0.0841368, 0.0813098
    0.0784420, 0.0755364, 0.0725962, 0.0696262, 0.0666327, 0.0636224, 0.0606016, -0.0637436
    -0.0601492, -0.0563668, -0.0523824, -0.0481823, -0.0437526, -0.0390796, -0.0341494, -0.0289481
    -0.0234621, -0.0176780, -0.0115977, -0.0052384, 0.0013820, 0.0082455, 0.0125032, 0.0077389
    0.0030834, -0.0014561, -0.0058727, -0.0101594, -0.0143091, -0.0183148, -0.0221695, -0.0258661
    -0.0293979, -0.0327624, -0.0359621, -0.0389996, -0.0418773, 0.1193166, 0.1212150, 0.1228393
    0.1241749, 0.1252072, 0.1259215, 0.1263033, 0.1263380, 0.1260110, 0.1253076, 0.1242140
    0.1227300, 0.1208703, 0.1186500, 0.1160843, -0.1185704, -0.1148212, -0.1108735, -0.1067269
    -0.1023809, -0.0978348, -0.0930883, -0.0881406, -0.0829914, -0.0776400, -0.0720863, -0.0663355
    -0.0603990, -0.0542886, -0.0480157, 0.0583250, 0.0564782, 0.0548263, 0.0533813, 0.0521553
    0.0511605, 0.0504090, 0.0499130, 0.0496845, 0.0497356, 0.0500779, 0.0507077, 0.0516058
    0.0527522, 0.0541270, 0.1353638, 0.1313381, 0.1272324, 0.1230490, 0.1187897, 0.1144566
    0.1100518, 0.1055772, 0.1010349, 0.0964268, 0.0917550, 0.0870218, 0.0822297, 0.0773811
    0.0724786, -0.0180711, -0.0229253, -0.0277300, -0.0324813, -0.0371753, -0.0418079, -0.0463752
    -0.0508733, -0.0552981, -0.0596458, -0.0639125, -0.0680959, -0.0721960, -0.0762126, -0.0801455
    0.1276658, 0.1281422, 0.1286489, 0.1291845, 0.1297478, 0.1303374, 0.1309519, 0.1315901
    0.1322506, 0.1329321, 0.1336332, 0.1343503, 0.1350780, 0.1358105, 0.1365422, 0.1341147
    0.1308563, 0.1273050, 0.1234552, 0.1193012, 0.1148372, 0.1100576, 0.1049567, 0.0995287
    0.0937679, 0.0876691, 0.0812383, 0.0744930, 0.0674512, 0.0601309, 0.0900934, 0.0884138
    0.0867445, 0.0850886, 0.0834493, 0.0818300, 0.0802338, 0.0786640, 0.0771239, 0.0756166
    0.0741453, 0.0727099, 0.0713072, 0.0699338, 0.0685862, 0.0413872, 0.0350636, 0.0287237
    0.0223717, 0.0160115, 0.0096474, 0.0032833, -0.0030765, -0.0094280, -0.0157671, -0.0220896
    -0.0283901, -0.0346618, -0.0408980, -0.0470918, 0.0755875, 0.0739173, 0.0718717, 0.0694406
    0.0666140, 0.0633818, 0.0597340, 0.0556606, 0.0511514, 0.0461965, 0.0407865, 0.0349304
    0.0286561, 0.0219922, 0.0149673, 0.1297014, 0.1303879, 0.1309192, 0.1312868, 0.1314823
    0.1314970, 0.1313227, 0.1309508, 0.1303729, 0.1295806, 0.1285656, 0.1273265, 0.1258690
    0.1241989, 0.1223223, -0.0027479, 0.0012134, 0.0050790, 0.0088355, 0.0124699, 0.0159688
    0.0193190, 0.0225073, 0.0255204, 0.0283451, 0.0309686, 0.0333890, 0.0356160, 0.0376592
    0.0395288, 0.0290004, 0.0302992, 0.0316568, 0.0330863, 0.0346009, 0.0362138, 0.0379380
    0.0397869, 0.0417735, 0.0439110, 0.0462122, 0.0486769, 0.0512924, 0.0540451, 0.0569216
    0.0448184, 0.0512294, 0.0576943, 0.0642108, 0.0707761, 0.0773878, 0.0840433, 0.0907400
    0.0974754, 0.1042470, 0.1110519, 0.1178836, 0.1247314, 0.1315844, 0.1384318, 0.0079080
    0.0043265, 0.0007314, -0.0028650, -0.0064505, -0.0100129, -0.0135401, -0.0170198, -0.0204398
    -0.0237880, -0.0270524, -0.0302289, -0.0333209, -0.0363325, -0.0392677, 0.1357616, 0.1397761
    0.1436628, 0.1474197, 0.1510451, 0.1545371, 0.1578940, 0.1611140, 0.1641951, 0.1671357
    0.1699338, 0.1725850, 0.1750826, 0.1774196, 0.1795891, 0.1128528, 0.1144198, 0.1158386
    0.1171095, 0.1182329, 0.1192093, 0.1200389, 0.1207222, 0.1212594, 0.1216511, 0.1218977
    0.1220020, 0.1219696, 0.1218062, 0.1215172, 0.1761363, 0.1778200, 0.1793493, 0.1807218
    0.1819351, 0.1829867, 0.1838742, 0.1845951, 0.1851470, 0.1855273, 0.1857340, 0.1857693
    0.1856408, 0.1853559, 0.1849222, -0.0491497, -0.0454618, -0.0415915, -0.0375284, -0.0332623
    -0.0287830, -0.0240801, -0.0191433, -0.0139624, -0.0085271, -0.0028278, 0.0031299, 0.0093246
    0.0157340, 0.0223362, 0.1469728, 0.1491036, 0.1511741, 0.1531834, 0.1551309, 0.1570156
    0.1588368, 0.1605937, 0.1622854, 0.1639111, 0.1654701, 0.1669597, 0.1683763, 0.1697156
    0.1709738, 0.3216147, 0.3118152, 0.3017543, 0.2914528, 0.2809313, 0.2702106, 0.2593112
    0.2482539, 0.2370593, 0.2257481, 0.2143409, 0.2028543, 0.1913016, 0.1796954, 0.1680488
    -0.0159183, -0.0107352, -0.0056755, -0.0007505, 0.0040286, 0.0086507, 0.0131043, 0.0173784
    0.0214616, 0.0253428, 0.0290110, 0.0324666, 0.0357209, 0.0387858, 0.0416731, -0.0254413
    -0.0274388, -0.0293219, -0.0310746, -0.0326807, -0.0341243, -0.0353892, -0.0364594, -0.0373189
    -0.0379516, -0.0383419, -0.0384855, -0.0383898, -0.0380625, -0.0375115, -0.0166281, -0.0149723
    -0.0134576, -0.0120888, -0.0108707, -0.0098081, -0.0089057, -0.0081684, -0.0076009, -0.0072079
    -0.0069941, -0.0069577, -0.0070906, -0.0073845, -0.0078309, -0.0174071, -0.0126844, -0.0078643
    -0.0029462, 0.0020701, 0.0071853, 0.0123996, 0.0177135, 0.0231274, 0.0286418, 0.0342568
    0.0399670, 0.0457610, 0.0516272, 0.0575540, -0.0985392, -0.0994117, -0.1002845, -0.1011639
    -0.1020565, -0.1029688, -0.1039072, -0.1048782, -0.1058883, -0.1069440, -0.1080513, -0.1092091
    -0.1104083, -0.1116396, -0.1128937, 0.0001530, 0.0035909, 0.0070450, 0.0105171, 0.0140092
    0.0175231, 0.0210608, 0.0246240, 0.0282147, 0.0318347, 0.0354860, 0.0391708, 0.0428918
    0.0466516, 0.0504531, -0.0819526, -0.0816026, -0.0811294, -0.0805304, -0.0798034, -0.0789457
    -0.0779550, -0.0768288, -0.0755645, -0.0741597, -0.0726123, -0.0709266, -0.0691139, -0.0671856
    -0.0651534, 0.0965162, 0.0928315, 0.0891501, 0.0854817, 0.0818362, 0.0782233, 0.0746527
    0.0711343, 0.0676778, 0.0642930, 0.0609896, 0.0577725, 0.0546423, 0.0515992, 0.0486437
    -0.2427283, -0.2398448, -0.2368635, -0.2337869, -0.2306173, -0.2273569, -0.2240082, -0.2205735
    -0.2170550, -0.2134551, -0.2097761, -0.2060230, -0.2022031, -0.1983238, -0.1943926, -0.1351105
    -0.1374491, -0.1394984, -0.1412510, -0.1426992, -0.1438354, -0.1446521, -0.1451416, -0.1452964
    -0.1451089, -0.1445720, -0.1436916, -0.1424869, -0.1409778, -0.1391840, -0.0198544, -0.0241394
    -0.0282630, -0.0322126, -0.0359753, -0.0395385, -0.0428895, -0.0460155, -0.0489037, -0.0515415
    -0.0539166, -0.0560280, -0.0578859, -0.0595013, -0.0608852, 0.1033334, 0.0997555, 0.0962746
    0.0929015, 0.0896467, 0.0865207, 0.0835341, 0.0806975, 0.0780214, 0.0755164, 0.0731926
    0.0710490, 0.0690733, 0.0672527, 0.0655744, -0.0997362, -0.1019782, -0.1039813, -0.1057214
    -0.1071745, -0.1083168, -0.1091242, -0.1095728, -0.1096387, -0.1092978, -0.1085273, -0.1073275
    -0.1057235, -0.1037410, -0.1014061, -0.0270366, -0.0233783, -0.0198873, -0.0165889, -0.0135084
    -0.0106710, -0.0081018, -0.0058263, -0.0038695, -0.0022567, -0.0010125, -0.0001434, 0.0003625
    0.0005178, 0.0003354, -0.0572062, -0.0531361, -0.0493332, -0.0458104, -0.0425804, -0.0396559
    -0.0370498, -0.0347749, -0.0328439, -0.0312696, -0.0300643, -0.0292248, -0.0287326, -0.0285681
    -0.0287122, 0.0384271, 0.0400259, 0.0414649, 0.0427437, 0.0438614, 0.0448175, 0.0456113
    0.0462421, 0.0467093, 0.0470122, 0.0471505, 0.0471296, 0.0469615, 0.0466583, 0.0462322
    0.0717728, 0.0695893, 0.0672396, 0.0647269, 0.0620541, 0.0592243, 0.0562403, 0.0531053
    0.0498221, 0.0463938, 0.0428236, 0.0391184, 0.0352894, 0.0313478, 0.0273048, -0.0450516
    -0.0419416, -0.0386771, -0.0352532, -0.0316651, -0.0279082, -0.0239776, -0.0198686, -0.0155764
    -0.0110964, -0.0064241, -0.0015652, 0.0034640, 0.0086470, 0.0139673, -0.0612851, -0.0675632
    -0.0737045, -0.0796916, -0.0855072, -0.0911338, -0.0965540, -0.1017504, -0.1067057, -0.1114025
    -0.1158238, -0.1199621, -0.1238200, -0.1274002, -0.1307057, -0.2006412, -0.1943896, -0.1878903
    -0.1811593, -0.1742131, -0.1670678, -0.1597397, -0.1522450, -0.1446002, -0.1368213, -0.1289246
    -0.1209250, -0.1128360, -0.1046710, -0.0964436, -0.1101506, -0.1094286, -0.1087262, -0.1080474
    -0.1073962, -0.1067766, -0.1061925, -0.1056480, -0.1051469, -0.1046933, -0.1042911, -0.1039389
    -0.1036309, -0.1033608, -0.1031222, -0.0820308, -0.0763831, -0.0706635, -0.0648856, -0.0590631
    -0.0532094, -0.0473381, -0.0414628, -0.0355971, -0.0297545, -0.0239484, -0.0181894, -0.0124847
    -0.0068417, -0.0012675, 0.0917091, 0.0912821, 0.0905308, 0.0894406, 0.0879973, 0.0861863
    0.0839933, 0.0814040, 0.0784038, 0.0749785, 0.0711144, 0.0668170, 0.0621115, 0.0570237
    0.0515798, -0.1294626, -0.1272798, -0.1249988, -0.1226242, -0.1201607, -0.1176130, -0.1149858
    -0.1122837, -0.1095114, -0.1066737, -0.1037752, -0.1008182, -0.0978032, -0.0947306, -0.0916005
    0.0030728, 0.0004540, -0.0022056, -0.0048990, -0.0076197, -0.0103606, -0.0131151, -0.0158763
    -0.0186375, -0.0213918, -0.0241325, -0.0268558, -0.0295605, -0.0322458, -0.0349107, -0.0715038
    -0.0802228, -0.0888249, -0.0972798, -0.1055570, -0.1136262, -0.1214571, -0.1290192, -0.1362821
    -0.1432156, -0.1497899, -0.1559936, -0.1618334, -0.1673172, -0.1724528, -0.0293459, -0.0276742
    -0.0259024, -0.0240231, -0.0220287, -0.0199119, -0.0176651, -0.0152810, -0.0127520, -0.0100708
    -0.0072302, -0.0042324, -0.0010891, 0.0021876, 0.0055856, -0.0198894, -0.0164613, -0.0130398
    -0.0096217, -0.0062041, -0.0027840, 0.0006417, 0.0040759, 0.0075217, 0.0109821, 0.0144599
    0.0179544, 0.0214613, 0.0249760, 0.0284940, -0.0632152, -0.0687483, -0.0741381, -0.0793737
    -0.0844447, -0.0893403, -0.0940500, -0.0985630, -0.1028687, -0.1069565, -0.1108161, -0.1144450
    -0.1178493, -0.1210351, -0.1240087, 0.1738959, 0.1710729, 0.1680760, 0.1649032, 0.1615524
    0.1580214, 0.1543082, 0.1504108, 0.1463269, 0.1420544, 0.1375917, 0.1329436, 0.1281220
    0.1231391, 0.1180071, -0.0365145, -0.0358539, -0.0351557, -0.0344178, -0.0336381, -0.0328145
    -0.0319450, -0.0310275, -0.0300599, -0.0290402, -0.0279663, -0.0268400, -0.0256666, -0.0244514
    -0.0232000, -0.0122952, -0.0037388, 0.0045537, 0.0125514, 0.0202236, 0.0275394, 0.0344680
    0.0409785, 0.0470402, 0.0526223, 0.0576949, 0.0622538, 0.0663209, 0.0699191, 0.0730716];

   // MatMul 'l1_base': W(4×16) + b(4)
   w5 : ARRAY[0..67] OF REAL :=
[0.0431468, -0.7218783, -0.7664040, 0.0446040, 0.6287033, -0.2051307, -0.3788366, 0.4265812
    -0.5566995, 0.4906082, -0.1110822, 0.1812111, 0.4454913, -0.3052935, -0.5214026, -0.7138628
    0.9783757, -1.8518010, -0.4568165, -1.1427149, -0.0874276, -0.7568773, 0.8611937, -0.0933256
    0.6472971, -1.0294341, 0.3256389, 0.2590011, -0.7163869, 0.5744135, 0.3259708, -0.5870056
    0.2935589, 0.9891618, 1.2448254, 0.7247065, -0.0131453, 0.8092904, 0.1742139, -0.9718143
    0.1236900, 0.7221795, -0.6175265, -1.0537282, 0.4511162, -0.5315267, 0.3452142, 0.2253288
    -1.2039654, 1.2277515, -0.3759507, 0.7626216, -0.6206948, 0.7239274, 0.0452536, 0.7874691
    -0.5805001, -0.4060238, 0.7050563, 0.3644256, -0.6624428, -0.3291764, -0.9541196, 0.6871611
    0.0, 0.0, 0.0, 0.0];

   // Total: 6 array blocks
   END_STRUCT;
BEGIN
END_DATA_BLOCK

FUNCTION "BsplineEval" : REAL
{ S7_Optimized_Access := 'FALSE' }
VERSION : 0.1
VAR_INPUT
    x : REAL;
    lut_grid : ARRAY[0..14] OF REAL;
    lut_table : ARRAY[0..14] OF REAL;
END_VAR
VAR_TEMP
    lo, hi, mid : INT;
    t, vlo, vhi : REAL;
END_VAR

BEGIN
    // Binary search for interval containing x
    lo := 0;
    hi := 14;
    WHILE hi - lo > 1 DO
        mid := lo + (hi - lo) / 2;
        IF x > lut_grid[mid] THEN lo := mid; ELSE hi := mid; END_IF;
    END_WHILE;

    // Linear interpolation: y = vlo*(1-t) + vhi*t
    vlo := lut_table[lo];
    vhi := lut_table[hi];
    t := (x - lut_grid[lo]) / (lut_grid[hi] - lut_grid[lo] + 1.0E-10);
    "BsplineEval" := vlo * (1.0 - t) + vhi * t;
END_FUNCTION

FUNCTION_BLOCK "NeuroPLC_Inference"
{ S7_Optimized_Access := 'FALSE' }
VERSION : 0.1
VAR_INPUT
    features : ARRAY[0..27] OF REAL;
END_VAR

VAR_OUTPUT
    fault_class : INT;
    confidence : REAL;
END_VAR

VAR
    i, j, k : INT;
    sum_val, max_val, t_val : REAL;
    v0 : ARRAY[0..27] OF REAL;
    v1 : ARRAY[0..27] OF REAL;
    v3 : ARRAY[0..15, 0..27] OF REAL;
    v2 : ARRAY[0..15] OF REAL;
    v4 : ARRAY[0..15] OF REAL;
    v5 : ARRAY[0..15] OF REAL;
    v7 : ARRAY[0..3, 0..15] OF REAL;
    v6 : ARRAY[0..3] OF REAL;
    v8 : ARRAY[0..3] OF REAL;
    v9 : ARRAY[0..3] OF REAL;
    lut_tmp : ARRAY[0..14] OF REAL;
END_VAR

BEGIN
    // ---- Input ----
    FOR i := 0 TO 27 DO
        v0[i] := features[i];
    END_FOR;

    // ---- l0_silu: SILU ----
    v1[0] := v0[0] / (1.0 + EXP(-v0[0]));
    v1[1] := v0[1] / (1.0 + EXP(-v0[1]));
    v1[2] := v0[2] / (1.0 + EXP(-v0[2]));
    v1[3] := v0[3] / (1.0 + EXP(-v0[3]));
    v1[4] := v0[4] / (1.0 + EXP(-v0[4]));
    v1[5] := v0[5] / (1.0 + EXP(-v0[5]));
    v1[6] := v0[6] / (1.0 + EXP(-v0[6]));
    v1[7] := v0[7] / (1.0 + EXP(-v0[7]));
    v1[8] := v0[8] / (1.0 + EXP(-v0[8]));
    v1[9] := v0[9] / (1.0 + EXP(-v0[9]));
    v1[10] := v0[10] / (1.0 + EXP(-v0[10]));
    v1[11] := v0[11] / (1.0 + EXP(-v0[11]));
    v1[12] := v0[12] / (1.0 + EXP(-v0[12]));
    v1[13] := v0[13] / (1.0 + EXP(-v0[13]));
    v1[14] := v0[14] / (1.0 + EXP(-v0[14]));
    v1[15] := v0[15] / (1.0 + EXP(-v0[15]));
    v1[16] := v0[16] / (1.0 + EXP(-v0[16]));
    v1[17] := v0[17] / (1.0 + EXP(-v0[17]));
    v1[18] := v0[18] / (1.0 + EXP(-v0[18]));
    v1[19] := v0[19] / (1.0 + EXP(-v0[19]));
    v1[20] := v0[20] / (1.0 + EXP(-v0[20]));
    v1[21] := v0[21] / (1.0 + EXP(-v0[21]));
    v1[22] := v0[22] / (1.0 + EXP(-v0[22]));
    v1[23] := v0[23] / (1.0 + EXP(-v0[23]));
    v1[24] := v0[24] / (1.0 + EXP(-v0[24]));
    v1[25] := v0[25] / (1.0 + EXP(-v0[25]));
    v1[26] := v0[26] / (1.0 + EXP(-v0[26]));
    v1[27] := v0[27] / (1.0 + EXP(-v0[27]));

